				CASHCODE_STATE.RESET:
				CASHCODE_STATE.DISABLE:
					IF NOT fl_disableCashCode THEN
						eStateCashCode := CASHCODE_STATE.INIT;
					END_IF
			END_CASE

		CCNET_STATE.SEND_RESET:
			_BUFFER_CLEAR(PT:=ADR(sReadBuff), SIZE:=SIZEOF((sReadBuff)));
			_BUFFER_CLEAR(PT:=ADR(sReadData), SIZE:=SIZEOF((sReadData)));
			_BUFFER_CLEAR(PT:=ADR(sWriteData), SIZE:=SIZEOF((sWriteData)));
			SET_RESET();
			xDone := FALSE;
			szReadData := 0;
			eStateCCNET := CCNET_STATE.SEND_COMMAND;
		
		CCNET_STATE.SEND_POLL:
			_BUFFER_CLEAR(PT:=ADR(sReadBuff), SIZE:=SIZEOF((sReadBuff)));
			_BUFFER_CLEAR(PT:=ADR(sReadData), SIZE:=SIZEOF((sReadData)));
			_BUFFER_CLEAR(PT:=ADR(sWriteData), SIZE:=SIZEOF((sWriteData)));
			fb_COMread
			(
				xExecute := TRUE,
				hCom := hCom,
				pBuffer := ADR(sReadData),
				szBuffer := SIZEOF(sReadData),
			);
			IF  fb_COMread.xDone THEN
				szReadData1 := fb_COMread.szSize;
				fb_COMread(xExecute:=FALSE);
				IF  szReadData1 = 0 THEN 
					eStateCCNET := CCNET_STATE.SEND_COMMAND;
				END_IF
			END_IF
		
			_BUFFER_CLEAR(PT:=ADR(sReadBuff), SIZE:=SIZEOF((sReadBuff)));
			_BUFFER_CLEAR(PT:=ADR(sReadData), SIZE:=SIZEOF((sReadData)));
			_BUFFER_CLEAR(PT:=ADR(sWriteData), SIZE:=SIZEOF((sWriteData)));
			SET_POLL();
			xDone := FALSE;
			szReadData := 0;

		CCNET_STATE.SEND_ENABLE_BILL_TYPES:
			_BUFFER_CLEAR(PT:=ADR(sReadBuff), SIZE:=SIZEOF((sReadBuff)));
			_BUFFER_CLEAR(PT:=ADR(sReadData), SIZE:=SIZEOF((sReadData)));
			_BUFFER_CLEAR(PT:=ADR(sWriteData), SIZE:=SIZEOF((sWriteData)));
			SET_ENABLE_BILL_TYPES();
			xDone := FALSE;
			szReadData := 0;
			eStateCCNET := CCNET_STATE.SEND_COMMAND;

		CCNET_STATE.SEND_NSC:
			_BUFFER_CLEAR(PT:=ADR(sReadBuff), SIZE:=SIZEOF((sReadBuff)));
			_BUFFER_CLEAR(PT:=ADR(sReadData), SIZE:=SIZEOF((sReadData)));
			_BUFFER_CLEAR(PT:=ADR(sWriteData), SIZE:=SIZEOF((sWriteData)));
			SET_NSC();
			xDone := FALSE;
			szReadData := 0;
			fb_COMwrite
			(
				xExecute := TRUE,
				hCom := hCom,
				pBuffer := ADR(sWriteData),
				szSize := szWriteDataLen
				//szSize := INT_TO_UINT(LEN(sWriteData))
			);
			IF fb_COMwrite.xError THEN
				xWriteError := TRUE;
				eStateCCNET := CCNET_STATE.POLLING_CYCLE_ENDS;
			END_IF
			IF fb_COMwrite.xDone THEN
				fb_COMwrite(xExecute:=FALSE);
				xWriteError := FALSE;
				eStateCCNET := CCNET_STATE.RESPONSE_DELAY;
			END_IF

		CCNET_STATE.SEND_ASC:
			_BUFFER_CLEAR(PT:=ADR(sReadBuff), SIZE:=SIZEOF((sReadBuff)));
			_BUFFER_CLEAR(PT:=ADR(sReadData), SIZE:=SIZEOF((sReadData)));
			_BUFFER_CLEAR(PT:=ADR(sWriteData), SIZE:=SIZEOF((sWriteData)));
			SET_ACK();
			xDone := FALSE;
			szReadData := 0;
			fb_COMwrite
			(
				xExecute := TRUE,
				hCom := hCom,
				pBuffer := ADR(sWriteData),
				szSize := szWriteDataLen
				//szSize := INT_TO_UINT(LEN(sWriteData))
			);
			IF fb_COMwrite.xError THEN
				xWriteError := TRUE;
				eStateCCNET := CCNET_STATE.POLLING_CYCLE_ENDS;
			END_IF
			IF fb_COMwrite.xDone THEN
				fb_COMwrite(xExecute:=FALSE);
				xWriteError := FALSE;
				eStateCCNET := CCNET_STATE.RESPONSE_DELAY;
			END_IF
			
		CCNET_STATE.SEND_COMMAND:
			fb_COMwrite
			(
				xExecute := TRUE,
				hCom := hCom,
				pBuffer := ADR(sWriteData),
				szSize := szWriteDataLen
				//szSize := INT_TO_UINT(LEN(sWriteData))
			);
			IF fb_COMwrite.xError THEN
				xWriteError := TRUE;
				eStateCCNET := CCNET_STATE.POLLING_CYCLE_ENDS;
			END_IF
			
			fb_TON_Poll(IN:=FALSE, PT:=c_tDelay);
			fb_TON_Poll(IN:=TRUE, PT:=c_tDelay);


			IF fb_COMwrite.xDone THEN
				fb_COMwrite(xExecute:=FALSE);
				xWriteError := FALSE;
				fb_TON_Write(IN:=FALSE, PT:=c_tTimeoutWrite);
				fb_TON_Write(IN:=TRUE, PT:=c_tTimeoutWrite);
				
				fb_TON_Read(IN:=FALSE, PT:=c_tTimeoutRead);
				fb_TON_Read(IN:=TRUE, PT:=c_tTimeoutRead);
				eStateCCNET := CCNET_STATE.WAIT_WRITE;
			END_IF

		CCNET_STATE.WAIT_WRITE:
			fb_TON_Write();
			IF fb_TON_Write.Q THEN
				eStateCCNET := CCNET_STATE.RECEIVE_RESPONSE;
				fb_TON_Write(IN:=FALSE);
			END_IF
		

		CCNET_STATE.RECEIVE_RESPONSE:
			fb_COMread
			(
				xExecute := TRUE,
				hCom := hCom,
				pBuffer := ADR(sReadData),
				szBuffer := SIZEOF(sReadData),
			);
			fb_TON_Read();
			IF fb_COMread.xError THEN
				xReadError := TRUE;
				eStateCCNET := CCNET_STATE.POLLING_CYCLE_ENDS;
			END_IF
			
			IF fb_COMread.xDone THEN
				xTimeout:=FALSE;
				CHECK_RESPONSE();
				fb_COMread(xExecute:=FALSE);
				IF xCorrectAnswer THEN
					GET_DATA_FROM_RESPONSE();
					fb_TON_Read(IN:=FALSE, PT:=c_tTimeoutRead);
					IF Status.moneyReceived > 0  THEN
						eStateCCNET := CCNET_STATE.WAIT_ENROLLMENT;
						sum := sum + Status.moneyReceived;
					ELSE
						eStateCCNET := CCNET_STATE.SEND_ASC;
					END_IF
					
					
				//ELSE
				//	//SET_NSC();
				//	eStateCCNET := CCNET_STATE.SEND_NSC;
				//	fb_TON_Read(IN:=FALSE, PT:=c_tTimeout);
				END_IF
				
			END_IF
			
			
			IF fb_TON_Read.Q THEN
				xTimeout := TRUE;
				eStateCCNET := CCNET_STATE.SEND_NSC;
				fb_TON_Read(IN:=FALSE, PT:=c_tTimeoutRead);
//				OUTPUTS_TO_ZERO();
//				eStateCCNET := CCNET_STATE.RESPONSE_DELAY;
			END_IF

		CCNET_STATE.WAIT_ENROLLMENT:
			IF Status.moneyReceived  = 0 THEN
				eStateCCNET := CCNET_STATE.SEND_ASC;				
			END_IF
 			
			
			
		
		CCNET_STATE.RESPONSE_DELAY:
//			fb_TON(IN:=FALSE, PT:=c_tDelay);
//			fb_TON(IN:=TRUE, PT:=c_tDelay);
			eStateCCNET := CCNET_STATE.POLLING_CYCLE_ENDS;
			
		CCNET_STATE.POLLING_CYCLE_ENDS:
			fb_TON_Poll();
			IF fb_TON_Poll.Q THEN
				fb_COMread (xExecute:=FALSE);
				fb_COMwrite(xExecute:=FALSE);
				xCorrectAnswer := FALSE;
				xDone := TRUE;
				fb_TON_Poll(IN:=FALSE);
				eStateCCNET := CCNET_STATE.IDLE;
			END_IF

	END_CASE
	ELSE
		xDone := FALSE;
		xCorrectAnswer := FALSE;
//		OUTPUTS_TO_ZERO();
		eStateCCNET := CCNET_STATE.IDLE;
END_IF

ACTION CHECK_RESPONSE:
IF fb_COMread.szSize >= 6 THEN
//sReadData := CONCAT(sReadData,sReadBuff);
// szReadData := szReadData + fb_COMread.szSize;
 
// IF szReadData > 6 THEN
	wCRC:=GetCRC16(ADR(sReadData),UDINT_TO_WORD(fb_COMread.szSize-2) );   // Получим CRC 

	sWriteData[4] := WORD_TO_BYTE(wCRC); //LSB FIrst
	sWriteData[5] := WORD_TO_BYTE(SHR(wCRC, 8));

 	IF wCRC>0 OR (sReadData[fb_COMread.szSize-2] = WORD_TO_BYTE(wCRC) AND sReadData[fb_COMread.szSize-1] = WORD_TO_BYTE(SHR(wCRC, 8)) ) THEN
		FOR i:=0 TO UDINT_TO_INT(fb_COMread.szSize - 3) DO
			sReadBuff[i]:=sReadData[i];
		END_FOR
		xCorrectAnswer := TRUE;
	END_IF 
	 
// END_IF
 (*
     if (CRC16[0] = FAnswer[FLengthAnswer-2]) and (CRC16[1] = FAnswer[FLengthAnswer-1])
    //ответ полный и CRC верный а значит 100 % что данные верны, положим их в дату
    then
      begin
        // 5 это 1 байт синхронизации, 1 байт адресс девайса, 1 байт - длина данных, 2 байт - CRC
        CopyMemory(@FData,@FAnswer[3],FLengthAnswer-5);
        FLengthData:=FLengthAnswer-5;
      end
    else begin
           SendNSC(); // Скажем купу что мы получили неверный ответ
           raise Exception.Create('Не верный CRC ответа.');
         end;
  end

 
	IF FIND(sReadData, '>') <> 0 AND FIND(sReadData, '$R') <>0 AND
		(FIND(sReadData, '$R') > FIND(sReadData, '>')) THEN
		sReadData:=MID(sReadData, FIND(sReadData, '$R') - FIND(sReadData, '>') + 1,
		FIND(sReadData, '>'));
		xCorrectAnswer:=TRUE;
	END_IF
	*)
END_IF
END_ACTION

ACTION GET_DATA_FROM_RESPONSE:

IF eStateCashCode = CASHCODE_STATE.POLL THEN
	Z1 := sReadData[3]; //sReadData[fb_COMread.szSize-2]
	IF sReadData[2] = 7 THEN
		Z2 := sReadData[4];
	ELSE 
		Z2 := 0;	
	END_IF
	
	msg := "------";
	CASE Z1 OF
		
		16#10: //Power Up
				msg := "Power Up";
		16#11: //Power Up with Bill in Validator
				msg := "Power Up with Bill in Validator";
		16#12: // Power Up with Bill in Stacker
				msg := "Power Up with Bill in Stacker";
		16#13: //Initialize
				msg := "Initialize";
		16#14: //Idling
				msg := "Idling";
		16#15: //Accepting
				msg := "Accepting";
		16#17: //Stacking
				msg := "Stacking";
		16#18: //Returning
				msg := "Returning";
		16#19: //Unit Disabled
				msg := "Unit Disabled";
				eStateCashCode := CASHCODE_STATE.DISABLE;
		16#1A: //Holding
				msg := "Holding";
		16#1B: //Device Busy
				msg := "Device Busy";
		
		16#80: //money escrow!
				msg := "money escrow";
			cacheCodeConvertByteToMoney := 0;
			
			CASE Z2 OF
			   2: cacheCodeConvertByteToMoney :=10;
			   3: cacheCodeConvertByteToMoney :=50;
			   4: cacheCodeConvertByteToMoney :=100;
			   5: cacheCodeConvertByteToMoney :=500;
			   6: cacheCodeConvertByteToMoney :=1000;
			   7: cacheCodeConvertByteToMoney :=5000;   
			END_CASE
			
		
		16#81: //money received!
				msg := "money received";
			cacheCodeConvertByteToMoney := 0;
			
			CASE Z2 OF
			   2: cacheCodeConvertByteToMoney :=10;
			   3: cacheCodeConvertByteToMoney :=50;
			   4: cacheCodeConvertByteToMoney :=100;
			   5: cacheCodeConvertByteToMoney :=500;
			   6: cacheCodeConvertByteToMoney :=1000;
			   7: cacheCodeConvertByteToMoney :=5000;   
			END_CASE
			// счётчики по номиналам
			CASE Z2 OF
			   2: 
				   Status.receivedBanknote10 := 1;
			   3: 
				   Status.receivedBanknote50 := 1;
			   4:
					Status.receivedBanknote100 := 1; 
			   5:
					Status.receivedBanknote500 := 1; 
			   6:
					Status.receivedBanknote1000 := 1; 
			   7:
					Status.receivedBanknote5000 := 1; 
			END_CASE				
			//Status.countBanknote := 1; // +=1?
			//sum := sum + cacheCodeConvertByteToMoney;
			//amountReceived := cacheCodeConvertByteToMoney;
			Status.moneyReceived := cacheCodeConvertByteToMoney;
	
		16#1C: //Generic rejecting code.	
					msg := "Generic rejecting code.";
			CASE Z2 OF
				16#60:	// Insertion error - Rejecting due TO Insertion
					msg := "Insertion error";
				16#61:	// Rejecting due to Magnetic - Dielectric error
					msg := "Rejecting due to Magnetic";
				16#62:	// Rejecting due to Remained bill in head - Previously inserted bill remains in head
					msg := "Rejecting due to Remained bill in head";
				16#63:	// Rejecting due to Multiplying - Compensation error/multiplying factor error
					msg := "Rejecting due to Multiplying";
				16#64:	//Rejecting due to Conveying - Bill transport error
					msg := "Rejecting due to Conveying";
				16#65:	//Rejecting due to Identification1 - Identification error
					msg := "Rejecting due to Identification1";
				16#66:	//Rejecting due to Verification - Verification error
					msg := "Rejecting due to Verification";
				16#67:	//Rejecting due to Optic - Optic Sensor error
					msg := "Rejecting due to Optic";
				16#68:	//Rejecting due to Inhibit - Return by “inhibit denomination” error
					msg := "Rejecting due to Inhibit";
				16#69:	//Rejecting due to Capacity - Capacitance error
					msg := "Rejecting due to Capacity";
				16#6A:	//Rejecting due to Operation - Operation error
					msg := "Rejecting due to Operation";
				16#6C:	//Rejecting due to Length - Length error
					msg := "Rejecting due to Length";

				16#92:	//Rejecting due to unrecognised barcode - Bill taken was treated as a barcode but no reliable data can be read from it.
					msg := "Rejecting due to unrecognised barcode";

				16#6D:	//Rejecting due to UV - Banknote UV properties do not meet the predefined criteria
					msg := "Rejecting due to UV";

				16#93:	//Rejecting due to incorrect number of characters in barcode - Barcode data was read (at list partially) but is inconsistent.
					msg := "Rejecting due to incorrect number of characters in barcode";

				16#94:	//Rejecting due to unknown barcode start sequence - Barcode was not read as no synchronization was established.
					msg := "Rejecting due to unknown barcode start sequence";

				16#95:	//Rejecting due to unknown barcode stop sequence - Barcode was read but trailing data is corrupt.
					msg := "Rejecting due to unknown barcode stop sequence";
			END_CASE

		16#41: // Drop Cassette Full - Drop Cassette full condition	
				msg := "Drop Cassette Full";
				;
		16#42: // Drop Cassette out of position - The Bill Validator has detected the drop cassette to be open or removed.
				msg := "Drop Cassette out of position";
				;
		16#43: // Validator Jammed - A bill(s) has jammed in the acceptance path.	
				msg := "Validator Jammed";
		16#44: // Drop Cassette Jammed - A bill has jammed in drop cassette.	
				msg := "Drop Cassette Jammed";
				;
		16#45: // Cheated - Bill Validator sends this event if the intentions of the user to deceive the Bill Validator are detected.
				msg := "Cheated";
				;

		16#46: // Pause  - When the user tries to insert a second bill when the previous bill is in the Bill Validator but has not been stacked. 
			   // Thus Bill Validator stops motion of the second bill until the second bill is removed.*				
				msg := "Pause";
				;

		16#47: // Generic Failure codes	
			CASE Z2 OF
				16#50:	// Stack Motor Failure - Drop Cassette Motor failure
					msg := "Stack Motor Failure";
				16#51:	// Transport Motor Speed Failure
					msg := "Transport Motor Speed Failure";
				16#52:	// Transport Motor Failure
					msg := "Transport Motor Failure";
				16#53:	// Aligning Motor Failure
					msg := "Aligning Motor Failure";
				16#54:	// Initial Cassette Status Failure
					msg := "Initial Cassette Status Failure";
				16#55:	// Optic Canal Failure
					msg := "Optic Canal Failure";
				16#56:	// Magnetic Canal Failure - Inductive sensor failed to respond
					msg := "Magnetic Canal Failure";
				16#5F:	// Capacitance Canal Failure - Capacitance sensor failed to respond
					msg := "Capacitance Canal Failure";
			END_CASE
		
	END_CASE //Z1
	
	// состояние и ошибка купюрника
	CASE Z1 OF
		16#10, 16#11, 16#12, 16#13, 16#14, 16#15, 16#17, 16#18, 16#19, 16#1A, 16#1B:
			Status.cashcodeStatus := Z1;
			Status.cashcodeError := 0;
		16#1C:
			Status.cashcodeStatus := Z2;
			Status.cashcodeError := 0;
		16#41, 16#42, 16#43, 16#44, 16#45, 16#46:
			Status.cashcodeStatus := 16#FF;
			Status.cashcodeError := Z1;
		16#47:
			Status.cashcodeStatus := 16#FF;
			Status.cashcodeError := Z2;
	END_CASE
	

	// снятие кассеты
	IF Z1 = 16#42 THEN
		Status.casetteDropped := 1;
	ELSE
		Status.casetteDropped := 0;
	END_IF
		
	// замятие
	IF Z1 = 16#43 OR Z1 = 16#44 THEN
		Status.banknoteJammed := 1;
	ELSE
		Status.banknoteJammed := 0;
	END_IF
END_IF
END_ACTION

METHOD GetCRC16 : WORD
///calculate CRC for buffer; receive full command buffer
//FUNCTION cacheCodeCRC : WORD
VAR_INPUT
	iCommandBuffer: POINTER TO BYTE;
	iCommandBufferSize: WORD;
END_VAR
VAR
	i: WORD;
	tmpCRC: WORD;
	j: WORD;
END_VAR
GetCRC16 := 0;
FOR i := 0 TO iCommandBufferSize - 1 DO
	tmpCRC := GetCRC16 XOR iCommandBuffer[i];
	FOR j := 0 TO 7 DO
		IF (tmpCRC AND WORD#16#0001) <> 0 THEN
			tmpCRC := SHR (tmpCRC,1);
			tmpCRC := tmpCRC XOR WORD#16#08408;
		ELSE
			tmpCRC := SHR (tmpCRC, 1);
		END_IF
	END_FOR;
	GetCRC16 := tmpCRC;	
END_FOR
END_METHOD

ACTION SET_ACK:
(*
sWriteData[0]:=16#23;
sAdress:=BYTE_TO_STRH(byAdress);
sWriteData[1]:=sAdress[0];
sWriteData[2]:=sAdress[1];
byCRC:=sWriteData[0]+sWriteData[1]+sWriteData[2];
sCRC:=BYTE_TO_STRH(byCRC);
sWriteData[3]:=sCRC[0];
sWriteData[4]:=sCRC[1];
sWriteData[5]:=16#D;
*)
//ClearCommand();

  //byLengthCommand:=6;
  szWriteDataLen := 6+0; //Длина всего пакета включая CRC

  sWriteData[0] := 02; // Синхронизационный байт
  sWriteData[1] := 03; // Адресс валидатора
  sWriteData[2] := UDINT_TO_BYTE(szWriteDataLen); //Длина всего пакета включая CRC
  sWriteData[3] := 16#00;   // Команда

  wCRC:=GetCRC16(ADR(sWriteData),UDINT_TO_WORD(szWriteDataLen-2) );   // Получим CRC
  sWriteData[4] := WORD_TO_BYTE(wCRC); //LSB FIrst
  sWriteData[5] := WORD_TO_BYTE(SHR(wCRC, 8));
  
(*
cacheCodeGetNoDataCommandBuffer[0] := BYTE#16#02; //Sync
cacheCodeGetNoDataCommandBuffer[1] := iPeripheralAddress; 
cacheCodeGetNoDataCommandBuffer[2] := BUFFER_SIZE; //full data length with crc 
cacheCodeGetNoDataCommandBuffer[3] := iCommandCode;

crc:=cacheCodeCrc(iCommandBuffer := ADR(cacheCodeGetNoDataCommandBuffer), iCommandBufferSize := BUFFER_SIZE);
cacheCodeGetNoDataCommandBuffer[4] := WORD_TO_BYTE(crc); //LSB FIrst
cacheCodeGetNoDataCommandBuffer[5] := WORD_TO_BYTE(SHR(crc, 8));
*)
  
//  if Length(Data) <> 0 // Если есть данные для пеердачи
//  then CopyMemory(@FCommand[4],@Data,Length(Data)); // Скопируем их все начиная с 5 байта
(*
  wCRC:=GetCRC16(sWriteData,6-2);   // Получим CRC
  CopyMemory(@CRC16,@CRCWord,2);             // Разабьем CRC на байты

  FCommand[FLengthCommand-2]:=CRC16[0];           // Подпишем нашу команду
  FCommand[FLengthCommand-1]:=CRC16[1];
*)
END_ACTION

ACTION SET_ENABLE_BILL_TYPES:
  szWriteDataLen := 6+6; //Длина всего пакета включая CRC

  sWriteData[0] := 02; // Синхронизационный байт
  sWriteData[1] := 03; // Адресс валидатора
  sWriteData[2] := UDINT_TO_BYTE(szWriteDataLen); //Длина всего пакета включая CRC
  sWriteData[3] := 16#34;   // Команда

  // примаемые купюры
  sWriteData[4] := 2#0000_0000;   // 
  sWriteData[5] := 2#0000_0000;   // 
  sWriteData[6] := 2#0001_1000;   //
  // депонируемые купюры (отложенные)
  sWriteData[7] := 2#1111_1111;   // 
  sWriteData[8] := 2#1111_1111;   // 
  sWriteData[9] := 2#1110_0111;   // 

  wCRC:=GetCRC16(ADR(sWriteData),UDINT_TO_WORD(szWriteDataLen-2) );   // Получим CRC
  sWriteData[10] := WORD_TO_BYTE(wCRC); //LSB FIrst
  sWriteData[11] := WORD_TO_BYTE(SHR(wCRC, 8));
END_ACTION

ACTION SET_NSC:
  szWriteDataLen := 6+0; //Длина всего пакета включая CRC

  sWriteData[0] := 02; // Синхронизационный байт
  sWriteData[1] := 03; // Адресс валидатора
  sWriteData[2] := UDINT_TO_BYTE(szWriteDataLen); //Длина всего пакета включая CRC
  sWriteData[3] := 16#FF;   // Команда

  wCRC:=GetCRC16(ADR(sWriteData),UDINT_TO_WORD(szWriteDataLen-2) );   // Получим CRC
  sWriteData[4] := WORD_TO_BYTE(wCRC); //LSB FIrst
  sWriteData[5] := WORD_TO_BYTE(SHR(wCRC, 8));
END_ACTION

ACTION SET_PAKET:

END_ACTION

ACTION SET_POLL:
  szWriteDataLen := 6+0; //Длина всего пакета включая CRC

  sWriteData[0] := 02; // Синхронизационный байт
  sWriteData[1] := 03; // Адресс валидатора
  sWriteData[2] := UDINT_TO_BYTE(szWriteDataLen); //Длина всего пакета включая CRC
  sWriteData[3] := 16#33;   // Команда

  wCRC:=GetCRC16(ADR(sWriteData),UDINT_TO_WORD(szWriteDataLen-2) );   // Получим CRC
  sWriteData[4] := WORD_TO_BYTE(wCRC); //LSB FIrst
  sWriteData[5] := WORD_TO_BYTE(SHR(wCRC, 8));
END_ACTION

ACTION SET_RESET:
  szWriteDataLen := 6+0; //Длина всего пакета включая CRC

  sWriteData[0] := 02; // Синхронизационный байт
  sWriteData[1] := 03; // Адресс валидатора
  sWriteData[2] := UDINT_TO_BYTE(szWriteDataLen); //Длина всего пакета включая CRC
  sWriteData[3] := 16#30;   // Команда

  wCRC:=GetCRC16(ADR(sWriteData),UDINT_TO_WORD(szWriteDataLen-2) );   // Получим CRC
  sWriteData[4] := WORD_TO_BYTE(wCRC); //LSB FIrst
  sWriteData[5] := WORD_TO_BYTE(SHR(wCRC, 8));

 // sWriteData[4] := 65;   // 
 // sWriteData[5] := 179;   //
END_ACTION

METHOD resetMoneyReceived : word
VAR_INPUT
END_VAR
Status.moneyReceived := 0;
END_METHOD

METHOD resetMoneyCnt
VAR_INPUT
END_VAR
Status.receivedBanknote10 := 0;
Status.receivedBanknote50 := 0;
Status.receivedBanknote100 := 0; 
Status.receivedBanknote500 := 0; 
Status.receivedBanknote1000 := 0; 
Status.receivedBanknote5000 := 0;
END_METHOD

END_FUNCTION_BLOCK

// CompWin/AppTerminalPost/Cash/_BUFFER_CLEAR
FUNCTION _BUFFER_CLEAR : BOOL
VAR_INPUT
	PT : POINTER TO BYTE;
	SIZE : UINT;
END_VAR

VAR
	ptw : POINTER TO DWORD;
	temp: DWORD;
	end, end32 : DWORD;
END_VAR

temp := pt;
end := temp + UINT_TO_DWORD(size);
end32 := end - 3;
WHILE (pt < end) AND ((temp AND 16#00000003) > 0) DO
pt^ := 0;
pt := pt + 1;
temp := temp + 1;
END_WHILE;
ptw := pt;
WHILE ptw < end32 DO
ptw^ := 0;
ptw := ptw + 4;
END_WHILE;
pt := ptw;
WHILE pt < end DO
pt^ := 0;
pt := pt + 1;
END_WHILE;
_BUFFER_CLEAR := TRUE;

END_FUNCTION

// CompWin/AppTerminalPost/Cash/ANALYZE_DATA
FUNCTION_BLOCK ANALYZE_DATA
VAR_INPUT
sData: STRING;
END_VAR
VAR CONSTANT
c_iMaxCanal: INT := 8;
END_VAR
VAR_OUTPUT
arValue: ARRAY [1..c_iMaxCanal] OF REAL;
END_VAR
VAR
aiSignPos: ARRAY [1..c_iMaxCanal+1] OF INT;
i,j: INT;
END_VAR

j:=1;
FOR i:=1 TO FIND(sData,'$R') DO
IF sData[i]=16#2B OR sData[i]=16#2D OR sData[i]=16#0D THEN
aiSignPos[j]:=i;
j:=j+1;
END_IF
END_FOR
FOR i:=1 TO c_iMaxCanal-1 DO
arValue[i]:= STRING_TO_REAL(MID(sData, aiSignPos[i+1] - aiSignPos[i], aiSignPos[i] + 1));
END_FOR
arValue[c_iMaxCanal]:=STRING_TO_REAL(
MID(sData, aiSignPos[c_iMaxCanal+1] - aiSignPos[c_iMaxCanal] - 2,
aiSignPos[i] + 1));

END_FUNCTION_BLOCK

// CompWin/AppTerminalPost/Cash/BYTE_TO_STRH
FUNCTION BYTE_TO_STRH : STRING(2)
VAR_INPUT
IN : BYTE;
END_VAR
VAR
temp : BYTE;
PT : POINTER TO BYTE;
END_VAR

PT := ADR(BYTE_TO_STRH);
temp := SHR(in,4);
IF temp <= 9 THEN temp := temp + 48; ELSE temp := temp + 55; END_IF;
PT^ := temp;
temp := in AND 2#00001111;
IF temp <= 9 THEN temp := temp + 48; ELSE temp := temp + 55; END_IF;
pt := pt + 1;
pt^ := temp;
pt := pt + 1;
pt^:= 0;

END_FUNCTION

// CompWin/AppTerminalPost/DevCoin/DeviceCoin
PROGRAM DeviceCoin
VAR
	amountReceived : WORD :=0;	
	_amountReceivedTemp: WORD := 0;

	_device: ccTalk;
	_deviceStatus: ccTalkStatus;
	_isInitialized: BOOL := FALSE;

	_isCollected: BOOL := FALSE;	// Признак проведённой инкассации для сброса количества купюр
//	countCoin: UINT := 0;		// Количество купюр в боксе

	uWarningCountCoin:		UINT;	//Предупредительное	количество монет в	приёмнике (шт)
	uMAXCountCoin:			UINT;	//Максимальное кол-во монет в CashBox (шт)

	message: STRING;
END_VAR

//В самом начале с помощью метода init задаём конфигурацию модуля
//Это делается один раз
IF NOT (_isInitialized) THEN
// инициализация монетника
//	_device.init(iComPort:= 3, iCoinTypes :=  COIN_10RUB OR COIN_5RUB OR COIN_2RUB OR COIN_1RUB);
	_device.init(iComPort:= 3, iCoinTypes :=  COIN_10RUB);
	_isInitialized :=  TRUE;
END_IF;

//проводим итерацию рабочего цикла и узнаём новый статус блока
_deviceStatus:=_device.iterateAndUpdateStatus();

IF (_deviceStatus.error = CCTALK_NO_ERROR AND NOT (_deviceStatus.busy) AND _deviceStatus.moneyReceived > 0) THEN
//	totalMoneyReceived := totalMoneyReceived + ccTalkStatus.moneyReceived;
	_amountReceivedTemp := _amountReceivedTemp + _deviceStatus.moneyReceived;
	//countCoin := countCoin + _deviceStatus.countCoin;

	PersistentVars.counterCoin10 := PersistentVars.counterCoin10 + _deviceStatus.receivedCoin10;

	// увеличить тотальные счётчики номиналов
	PersistentVars.totalCoin10 := PersistentVars.totalCoin10 + _deviceStatus.receivedCoin10;
END_IF

// если внешней программой была обработана сумма, то перенести принятую сумму в прееменную для внешенй обработки
IF(amountReceived = 0 AND _amountReceivedTemp > 0)THEN
	amountReceived := _amountReceivedTemp;
	_amountReceivedTemp := 0;
END_IF

// если внешней программой был сброшен счётчик купюр, то сбросить его внутри
IF(_isCollected)THEN
	//countCoin := 0;
(*	// Coin: m1=7; m2=8; m5=9; m10=10;
	message := 'Coin: ';
	message := CONCAT(message, 'm1=');
	message := CONCAT(message, WORD_TO_STRING(DeviceCoin.GetCounterCoin(1)));
	message := CONCAT(message, '; ');
	
	message := CONCAT(message, 'm2=');
	message := CONCAT(message, WORD_TO_STRING(DeviceCoin.GetCounterCoin(2)));
	message := CONCAT(message, '; ');
	
	message := CONCAT(message, 'm5=');
	message := CONCAT(message, WORD_TO_STRING(DeviceCoin.GetCounterCoin(5)));
	message := CONCAT(message, '; ');
	
	message := CONCAT(message, 'm10=');
	message := CONCAT(message, WORD_TO_STRING(DeviceCoin.GetCounterCoin(10)));
	message := CONCAT(message, ';');
	
	PersistentVars.messageCollectCoin := message;
*)

	// запомнить значения счётчиков
	// только если было начало инкассации и счётчики ещё не сброшены
	// (защита от повторного нажатия кнопок инкассации)
	IF(PersistentVars.counterBefCollectCoin10 = 0) THEN
		PersistentVars.counterBefCollectCoin10 := PersistentVars.counterCoin10;
	END_IF
		
	// сбросить значения
	PersistentVars.counterCoin10 := 0;

	_isCollected := FALSE;
END_IF

// Вернуть во вне принятую сумму, 
// затем сбросить сумму для записывания следующих принятий
METHOD PUBLIC GetReceived : WORD
GetReceived := amountReceived;

amountReceived := 0;
END_METHOD

METHOD PUBLIC DbgInCoin : BYTE
VAR_INPUT
END_VAR
VAR
	received: WORD := 0;
END_VAR
received := DBG_PRG.GetInCoin();
IF(received > 0)THEN
	_amountReceivedTemp := _amountReceivedTemp + received;
	//countCoin := countCoin + 1;
END_IF
END_METHOD

METHOD PUBLIC CollectCash : UINT
VAR_INPUT
END_VAR
// выстаитьВыставить признка необходимости сброса счётчика монет
_isCollected := TRUE;
END_METHOD

METHOD GetCounterCoin : UINT
VAR_INPUT
	// номинал
	nom: INT;
END_VAR
GetCounterCoin := 0;

CASE nom OF
	0:
		GetCounterCoin := PersistentVars.counterCoin10;
	10:
		GetCounterCoin := PersistentVars.counterCoin10;
END_CASE
END_METHOD

END_PROGRAM

// CompWin/AppTerminalPost/DevCoin/ccTalk
FUNCTION_BLOCK ccTalk
VAR CONSTANT
//	COM_PORT : BYTE := 2;  //use com2
	CCTALK_SLAVE_ID : BYTE := 2; //destination id
	CCTALK_MASTER_ID :BYTE := 1;
	
	CCTALK_COMMAND_RESET : BYTE := 1;  //reset command id
	
	CCTALK_COMMAND_MODIFY_INHIBIT_STATUS : BYTE :=  231; // modify inhibit status command id

	
	CCTALK_COMMAND_MODIFY_MASTER_INHIBIT_STATUS : BYTE :=  228; // modify inhibit status command id
	MODIFY_MASTER_INHIBIT_STATUS_COMMAND_DATA : ARRAY[0..0] OF BYTE := [1];
	
	//program states
	CCTALK_INIT_STATE : BYTE :=0;
	CCTALK_FATAL_ERROR_STATE : BYTE :=1;
	CCTALK_DONE_STATE : BYTE :=2;
	CCTALK_RESET_STATE : BYTE :=3;
	CCTALK_POLL_STATE: BYTE :=4;
	CCTALK_WAIT_STATE : BYTE :=5;
	CCTALK_DO_NOTHING_STATE: BYTE :=6;
	CCTALK_MODIFY_INHIBIT_STATUS_STATE: BYTE :=7;
	CCTALK_MODIFY_MASTER_INHIBIT_STATUS_STATE: BYTE :=8;
	CCTALK_READ_BUFFERED_CREDIT_STATE: BYTE :=9;
	
	CCTALK_CLOSE_COM_STATE : BYTE :=10;
	

END_VAR


VAR	

	RESET_TRYCOUNT_DELAY : TIME := T#1000MS; //delay between reset tries	
	POLL_DELAY : TIME := T#200MS;

	//cachecode program states
	state : BYTE := CCTALK_INIT_STATE;
	
	error: CCTALK_ERROR := CCTALK_INIT_PROC_NOT_CALLED;
	
	
	
	//com parameters
	ccTalkComParams : ARRAY [1..7] OF COM.PARAMETER := [     
		(udiParameterId := COM.CAA_Parameter_Constants.udiPort, udiValue := 0),  // COM порт
		(udiParameterId := COM.CAA_Parameter_Constants.udiBaudrate, udiValue := 9600),
		(udiParameterId := COM.CAA_Parameter_Constants.udiParity,udiValue := INT_TO_UDINT(COM.PARITY.NONE)),
	    (udiParameterId := COM.CAA_Parameter_Constants.udiStopBits,udiValue := INT_TO_UDINT(COM.STOPBIT.ONESTOPBIT)),
		(udiParameterId := COM.CAA_Parameter_Constants.udiTimeout, udiValue := 0),
		(udiParameterId := COM.CAA_Parameter_Constants.udiByteSize, udiValue := 8),
		(udiParameterId := COM.CAA_Parameter_Constants.udiBinary,udiValue := 0)
	];
	
	ccTalkOpen : COM.Open;
	ccTalkClose : COM.Close;
	openedHCom : CAA.HANDLE := 0;
	portOpened : BOOL := FALSE;
	
	simpleCommand : ccTalkSimpleCommand;
	readBufferedCreditCommand : ccTalkReadBufferedCreditCommand;

	
	
	waitTimer : TON;

	
	test:BYTE:=2;
	
	modifyInhibitStatusCommandData : ARRAY[0..1] OF BYTE ;
	
	moneyReceived : UINT := 0;
	coinsRejected : UINT := 0;
	
	receivedCoin1  : UINT := 0;
	receivedCoin2  : UINT := 0;
	receivedCoin5  : UINT := 0;
	receivedCoin10 : UINT := 0;
	// количество монет в боксе
	countCoin: UINT := 0;	
	
	
	b_cctalk_close_enable:  BOOL := FALSE;
END_VAR

METHOD init
VAR_INPUT
	iComPort: BYTE;
	///or`d  enabled coin types
	iCoinTypes: UINT := 0;
END_VAR
//init method called -> reset error flags
state := CCTALK_INIT_STATE;
error := CCTALK_NO_ERROR;

ccTalkComParams[1].udiValue := iComPort;
modifyInhibitStatusCommandData[0] := UINT_TO_BYTE(SHR(iCoinTypes, 8));
modifyInhibitStatusCommandData[1] := UINT_TO_BYTE(iCoinTypes);
END_METHOD

METHOD iterateAndUpdateStatus : ccTalkStatus
//waiting between cycle
	
coinsRejected := 0;
moneyReceived :=0;
countCoin := 0;

receivedCoin1 := 0;
receivedCoin2 := 0;
receivedCoin5 := 0;
receivedCoin10 := 0;

IF waitTimer.IN  THEN
	waitTimer(IN:= TRUE);
	IF NOT (waitTimer.Q) THEN
		iterateAndUpdateStatus.busy := simpleCommand.xExecute OR readBufferedCreditCommand.xExecute;
		iterateAndUpdateStatus.error := error;
		iterateAndUpdateStatus.moneyReceived := moneyReceived;
		iterateAndUpdateStatus.coinsRejected := coinsRejected ;
		
		iterateAndUpdateStatus.receivedCoin1 := receivedCoin1;
		iterateAndUpdateStatus.receivedCoin2 := receivedCoin2;
		iterateAndUpdateStatus.receivedCoin5 := receivedCoin5;
		iterateAndUpdateStatus.receivedCoin10 := receivedCoin10;
		
		
		RETURN;
	ELSE
		waitTimer(IN:=FALSE);	
	END_IF
END_IF


CASE state OF
	CCTALK_INIT_STATE:
		ccTalkOpen (xExecute := TRUE, 
				usiListLength := UINT_TO_USINT(SIZEOF(ccTalkComParams)/SIZEOF(COM.PARAMETER)),
				pParameterList:= ADR(ccTalkComParams)			
		);
		openedHCom := ccTalkOpen.hCom;
		IF ccTalkOpen.xError THEN
			ccTalkOpen (xExecute := FALSE);
			portOpened := FALSE;
			state := CCTALK_FATAL_ERROR_STATE;  
			error := CCTALK_OPEN_ERROR;
		END_IF;
		
		IF ccTalkOpen.xDone THEN
			ccTalkOpen (xExecute := FALSE);
			portOpened := TRUE;
			state := CCTALK_RESET_STATE;
			error := CCTALK_NO_ERROR;
		END_IF;
	CCTALK_RESET_STATE:
		simpleCommand(xExecute:=TRUE, hCom := openedHCom, xSourceId := CCTALK_MASTER_ID, 
					xDestinationId := CCTALK_SLAVE_ID, xCommand:=CCTALK_COMMAND_RESET, xCommandDataSize:=0 );
		
		IF simpleCommand.xDone THEN
			state := CCTALK_MODIFY_INHIBIT_STATUS_STATE;
			waitTimer(IN:= TRUE, PT := POLL_DELAY);
		END_IF
		
		//retry reset
		IF simpleCommand.xError THEN   
			state := CCTALK_CLOSE_COM_STATE;
			//state := CCTALK_RESET_STATE;
			waitTimer(IN:= TRUE, PT := RESET_TRYCOUNT_DELAY);
		END_IF
	CCTALK_CLOSE_COM_STATE:
		state := CCTALK_RESET_STATE;
		IF b_cctalk_close_enable THEN
			IF portOpened THEN
			  ccTalkClose(xExecute:=TRUE, hCom := openedHCom);
			  IF ccTalkClose.xError THEN
				portOpened := FALSE;
				ccTalkClose(xExecute:=FALSE);
				state := CCTALK_INIT_STATE;  
				error := CCTALK_OPEN_ERROR;
			  END_IF;
			  IF ccTalkClose.xDone THEN
				portOpened := FALSE;
				ccTalkClose(xExecute:=FALSE);
				state := CCTALK_INIT_STATE;
			  END_IF;
			ELSE		  
				state := CCTALK_INIT_STATE;
			END_IF;
	
		END_IF

	
	CCTALK_MODIFY_INHIBIT_STATUS_STATE: //enable coin types
		simpleCommand(xExecute:=TRUE, hCom := openedHCom, xSourceId := CCTALK_MASTER_ID, 
					 xDestinationId := CCTALK_SLAVE_ID, xCommand:=CCTALK_COMMAND_MODIFY_INHIBIT_STATUS, xCommandData:=
					 ADR(modifyInhibitStatusCommandData), xCommandDataSize := UINT_TO_BYTE(SIZEOF(modifyInhibitStatusCommandData))
					);
		
		IF simpleCommand.xDone THEN
			state := CCTALK_MODIFY_MASTER_INHIBIT_STATUS_STATE;
		END_IF
		
		//retry reset
		IF simpleCommand.xError THEN    
			state := CCTALK_RESET_STATE;
			waitTimer(IN:= TRUE, PT := POLL_DELAY);
		END_IF

	CCTALK_MODIFY_MASTER_INHIBIT_STATUS_STATE: //enable master inhibit
		simpleCommand(xExecute:=TRUE, hCom := openedHCom, xSourceId := CCTALK_MASTER_ID, 
					 xDestinationId := CCTALK_SLAVE_ID, xCommand:=CCTALK_COMMAND_MODIFY_MASTER_INHIBIT_STATUS, xCommandData:=
					 ADR(MODIFY_MASTER_INHIBIT_STATUS_COMMAND_DATA), xCommandDataSize := UINT_TO_BYTE(SIZEOF(MODIFY_MASTER_INHIBIT_STATUS_COMMAND_DATA))
					);
		
		IF simpleCommand.xDone THEN
			state := CCTALK_READ_BUFFERED_CREDIT_STATE;
		END_IF
		
		//retry reset
		IF simpleCommand.xError THEN    
			state := CCTALK_RESET_STATE;
			waitTimer(IN:= TRUE, PT := POLL_DELAY);
		END_IF	

	CCTALK_READ_BUFFERED_CREDIT_STATE: //
		readBufferedCreditCommand(xExecute:=TRUE, hCom := openedHCom, xSourceId := CCTALK_MASTER_ID, 
					 xDestinationId := CCTALK_SLAVE_ID);
		
		IF readBufferedCreditCommand.xDone THEN
			moneyReceived :=  readBufferedCreditCommand.xMoneyAccepted;
			coinsRejected := readBufferedCreditCommand.xCoinsRejected;
			countCoin := readBufferedCreditCommand.xCoinsAccepted;
			
			receivedCoin1 := readBufferedCreditCommand.xReceivedCoin1;
			receivedCoin2 := readBufferedCreditCommand.xReceivedCoin2;
			receivedCoin5 := readBufferedCreditCommand.xReceivedCoin5;
			receivedCoin10 := readBufferedCreditCommand.xReceivedCoin10;
			
			state := CCTALK_READ_BUFFERED_CREDIT_STATE;
			waitTimer(IN:= TRUE, PT := POLL_DELAY);
		END_IF
		
		//retry reset
		IF readBufferedCreditCommand.xError THEN    
			state := CCTALK_RESET_STATE;
			waitTimer(IN:= TRUE, PT := POLL_DELAY);
		END_IF			
		

	
	
	CCTALK_FATAL_ERROR_STATE:
		state := CCTALK_CLOSE_COM_STATE;
	
//	CCTALK_DONE_STATE:  //all work is done, free resources
//		ccTalkOpen(xExecute := FALSE);
//		state := CCTALK_DO_NOTHING_STATE;
//						
//	CCTALK_DO_NOTHING_STATE:
END_CASE


iterateAndUpdateStatus.busy := simpleCommand.xExecute OR readBufferedCreditCommand.xExecute;
iterateAndUpdateStatus.error := error;
iterateAndUpdateStatus.moneyReceived := moneyReceived;
iterateAndUpdateStatus.coinsRejected := coinsRejected ;

iterateAndUpdateStatus.countCoin := countCoin;
iterateAndUpdateStatus.receivedCoin1 := receivedCoin1;
iterateAndUpdateStatus.receivedCoin2 := receivedCoin2;
iterateAndUpdateStatus.receivedCoin5 := receivedCoin5;
iterateAndUpdateStatus.receivedCoin10 := receivedCoin10;
END_METHOD

END_FUNCTION_BLOCK

// CompWin/AppTerminalPost/DevCoin/ccTalkSimpleCommand
///command with  no-data ack
FUNCTION_BLOCK ccTalkSimpleCommand
VAR CONSTANT
	STATE_INITIAL: BYTE := 0;
	STATE_WAIT_ACK: BYTE := 1;
	STATE_FATAL_ERROR: BYTE := 3;
	COMMAND_EXPECTED_ANSWER_SIZE: BYTE := 5;
	///maximum size of command data 
	COMMAND_DATA_SIZE_MAX: BYTE := 5;
	COMMAND_DATA_OFFSET: BYTE := 4;
	///? 
END_VAR
VAR_INPUT
	hCom: CAA.HANDLE;
	xExecute: BOOL := FALSE;
	///device address
	xDestinationId: BYTE := 2;
	///master address, default = 1;
	xSourceId: BYTE := 1;
	xCommand: BYTE;
	xCommandData: POINTER TO BYTE;
	xCommandDataSize: BYTE := 0;
END_VAR
VAR_OUTPUT
	xDone: BOOL := FALSE;
	xError: BOOL := FALSE;
	xTimeout: BOOL := FALSE;
END_VAR
VAR
	TIMEOUT: TIME := TIME#200MS;
	///buffer for command
	commandBuffer: ARRAY[0..(4 + COMMAND_DATA_SIZE_MAX)] OF BYTE;
	///size enough for echo and answer
	//readBuffer: ARRAY[0..((4 + COMMAND_DATA_SIZE_MAX) + COMMAND_EXPECTED_ANSWER_SIZE)] OF BYTE;
	readBuffer: ARRAY[0..255] OF BYTE;
	///timeout timer (timeout value - ????)
	waitingACKtimeout: TON;
	localState: BYTE := STATE_INITIAL;
	ccTalkCodeWrite: COM.Write;
	ccTalkCodeRead: COM.Read;
	bufferReaded: CAA.SIZE := 0;
	bufferFullLen: BYTE := 5;
	///full answer size with echo
	fullAnswerSize: BYTE;
	commandCode: INT;
	crc: BYTE;
END_VAR

CASE localState OF 
	STATE_INITIAL:
		IF xExecute THEN
			xDone := FALSE;
			xError := FALSE;
			xTimeout := FALSE;
			IF NOT ccTalkCodeWrite.xExecute THEN
				bufferFullLen := 5 + xCommandDataSize;
				fullAnswerSize := bufferFullLen + COMMAND_EXPECTED_ANSWER_SIZE;
				commandBuffer[0] := xDestinationId;
				commandBuffer[1] := xCommandDataSize; //data size 
				commandBuffer[2] := xSourceId;  // master address
				commandBuffer[3] := xCommand; //command code
				IF xCommandDataSize > 0 THEN
					MEM.MemMove(pSource := xCommandData, pDestination := ADR(commandBuffer) + COMMAND_DATA_OFFSET, uiNumberOfBytes := xCommandDataSize);
				END_IF;
				commandBuffer[bufferFullLen - 1] := ccTalkCRC(ADR(commandBuffer), bufferFullLen); //command code
			END_IF
			ccTalkCodeWrite(xExecute := TRUE,hCom:= hCom, pBuffer:= ADR(commandBuffer), szSize:= bufferFullLen);
			IF ccTalkCodeWrite.xError THEN
				xError := TRUE;
				xExecute := FALSE;
				xCommandDataSize :=0;
				localState := STATE_INITIAL;
				ccTalkCodeWrite(xExecute := FALSE);
				RETURN;
			END_IF
		
			// if the writing process is completed the reading process can be started
			IF ccTalkCodeWrite.xDone THEN
				localState := STATE_WAIT_ACK;
				bufferReaded := 0;
				xCommandDataSize :=0;
				ccTalkCodeWrite(xExecute := FALSE);
				waitingACKtimeout(IN:=FALSE); 
				waitingACKtimeout(IN:=TRUE, PT:=TIMEOUT);  //timeout value ?
			END_IF			
		END_IF
		//waiting ACK
	STATE_WAIT_ACK:
		waitingACKtimeout(IN:=TRUE, PT:=TIMEOUT);  //timeout value ?
		IF waitingACKTimeout.Q THEN  //timeout is over..
			xError := TRUE;
			xExecute := FALSE;
			xTimeout := TRUE;
			localState := STATE_INITIAL;
			ccTalkCodeRead(xExecute := FALSE);
		ELSE
			ccTalkCodeRead(xExecute := TRUE,hCom:= hCom, pBuffer:= ADR(readBuffer) + bufferReaded, szBuffer:= SIZEOF(readBuffer)- bufferReaded);
			IF ccTalkCodeRead.xError THEN
				xError := TRUE;
				xExecute := FALSE;
				ccTalkCodeRead(xExecute := FALSE);
				localState := STATE_INITIAL;
			END_IF
			//After completion the size of the written bytes are saved
			IF 	ccTalkCodeRead.xDone THEN
				bufferReaded := bufferReaded + ccTalkCodeRead.szSize;
				IF bufferReaded >= fullAnswerSize THEN  //try to recognize command
					//MEM.MemMove(pSource:=ADR(readBuffer) + bufferFullLen, pDestination:=ADR(readBuffer), uiNumberOfBytes:=COMMAND_EXPECTED_ANSWER_SIZE); //move data to begin
					ccTalkCodeRead(xExecute := FALSE);
					crc := ccTalkCRC(iCommandBuffer := ADR(readBuffer), iCommandBufferSize:=COMMAND_EXPECTED_ANSWER_SIZE);
					//ALL OK
					IF (crc = readBuffer[COMMAND_EXPECTED_ANSWER_SIZE -1]) THEN
						//ack format :  [ destination, 0, source, 0, crc ] 
						IF readBuffer[0] = xSourceId AND readBuffer[1] = 0 AND readBuffer[2] = xDestinationId AND readBuffer[3] = 0 THEN 
							xExecute := FALSE;
							xDone := TRUE;
							localState := STATE_INITIAL;
						ELSE 
							bufferReaded := 0;  //try to wait buffer with proper fields
						END_IF
					ELSE
						xError := TRUE;
						xExecute := FALSE;
						localState := STATE_INITIAL;
					END_IF

				END_IF

			END_IF			
		END_IF
		
END_CASE

END_FUNCTION_BLOCK

// CompWin/AppTerminalPost/DevCoin/ccTalkCRC
///calculate CRC for buffer; receive full command buffer
FUNCTION ccTalkCRC : BYTE
VAR_INPUT
	iCommandBuffer: POINTER TO BYTE;
	iCommandBufferSize: WORD;
END_VAR
VAR
	i: WORD;
END_VAR

ccTalkCRC := 0;
FOR i := 0 TO iCommandBufferSize - 2 DO
	ccTalkCrc := ccTalkCrc + iCommandBuffer[i];
END_FOR
ccTalkCRC:= 255 - ccTalkCRC;
ccTalkCRC:=ccTalkCRC + 1;

END_FUNCTION

// CompWin/AppTerminalPost/DevCoin/ccTalkReadBufferedCreditCommand
///ReadBufferedCreditCommand (229).
FUNCTION_BLOCK ccTalkReadBufferedCreditCommand
VAR CONSTANT
	STATE_INITIAL: BYTE := 0;
	STATE_WAIT_ACK: BYTE := 1;
	STATE_FATAL_ERROR: BYTE := 3;
	COMMAND_EXPECTED_ANSWER_SIZE: BYTE := 16;
	COMMAND_EXPECTED_DATA_SIZE: BYTE := 11;
	///? 
	TIMEOUT: TIME := TIME#200ms;
END_VAR
VAR_INPUT
	hCom: CAA.HANDLE;
	xExecute: BOOL := FALSE;
	///device address
	xDestinationId: BYTE := 2;
	///master address, default = 1;
	xSourceId: BYTE := 1;
END_VAR
VAR_OUTPUT
	xDone: BOOL := FALSE;
	xError: BOOL := FALSE;
	xTimeout: BOOL := FALSE;
	///Total events since reset
	xEvents: BYTE := 0;
	xEventsTable: ARRAY[0..5] OF ccTalkEvent;
	///Money accepted since last poll
	xMoneyAccepted: BYTE := 0;
	///Coins rejected since last poll
	xCoinsRejected: BYTE := 0;
	///Coins accepted since last poll
	xCoinsAccepted : BYTE :=0;
	
	//Coins 1 ruble accepted since last poll
	xReceivedCoin1 : BYTE := 0;
	//Coins 2 ruble accepted since last poll
	xReceivedCoin2 : BYTE := 0;
	//Coins 5 ruble accepted since last poll
	xReceivedCoin5 : BYTE := 0;
	//Coins 10 ruble accepted since last poll
	xReceivedCoin10 : BYTE := 0;
END_VAR
VAR
	///last events
	lastEvents: BYTE := 0;
	///buffer for command
	commandBuffer: ARRAY[0..4] OF BYTE;
	///size enough for echo and answer
	//readBuffer: ARRAY[0..(4 + COMMAND_EXPECTED_ANSWER_SIZE)] OF BYTE;
	readBuffer: ARRAY[0..255] OF BYTE;
	///timeout timer (timeout value - ????)
	waitingACKtimeout: TON;
	localState: BYTE := STATE_INITIAL;
	ccTalkCodeWrite: COM.Write;
	ccTalkCodeRead: COM.Read;
	bufferReaded: CAA.SIZE := 0;
	bufferFullLen: BYTE := 5;
	///full answer size with echo
	fullAnswerSize: BYTE;
	commandCode: INT;
	crc: BYTE;
END_VAR

CASE localState OF 
	STATE_INITIAL:
		IF xExecute THEN
			xDone := FALSE;
			xError := FALSE;
			xTimeout := FALSE;
			IF NOT ccTalkCodeWrite.xExecute THEN
				xMoneyAccepted := 0;
				xCoinsRejected :=0;
				xCoinsAccepted :=0;
				bufferFullLen := 5;
				
				xReceivedCoin1 := 0;
				xReceivedCoin2 := 0;
				xReceivedCoin5 := 0;
				xReceivedCoin10 := 0;
				
				
				fullAnswerSize := bufferFullLen + COMMAND_EXPECTED_ANSWER_SIZE;
				commandBuffer[0] := xDestinationId;
				commandBuffer[1] := 0; //data size 
				commandBuffer[2] := xSourceId;  // master address
				commandBuffer[3] := 229; //command code
				commandBuffer[bufferFullLen - 1] := ccTalkCRC(ADR(commandBuffer), bufferFullLen); //command code
			END_IF
			ccTalkCodeWrite(xExecute := TRUE,hCom:= hCom, pBuffer:= ADR(commandBuffer), szSize:= bufferFullLen);
			IF ccTalkCodeWrite.xError THEN
				xError := TRUE;
				xExecute := FALSE;
				localState := STATE_INITIAL;
				ccTalkCodeWrite(xExecute := FALSE);
				RETURN;
			END_IF
		
			// if the writing process is completed the reading process can be started
			IF ccTalkCodeWrite.xDone THEN
				localState := STATE_WAIT_ACK;
				bufferReaded := 0;
				ccTalkCodeWrite(xExecute := FALSE);
				waitingACKtimeout(IN:=FALSE); 
				waitingACKtimeout(IN:=TRUE, PT:=TIMEOUT);  //timeout value ?
			END_IF			
		END_IF
		//waiting ACK
	STATE_WAIT_ACK:
		waitingACKtimeout(IN:=TRUE, PT:=TIMEOUT);  //timeout value ?
		IF waitingACKTimeout.Q THEN  //timeout is over..
			xError := TRUE;
			xExecute := FALSE;
			xTimeout := TRUE;
			localState := STATE_INITIAL;
			ccTalkCodeRead(xExecute := FALSE);
		ELSE
			ccTalkCodeRead(xExecute := TRUE,hCom:= hCom, pBuffer:= ADR(readBuffer) + bufferReaded, szBuffer:= SIZEOF(readBuffer)- bufferReaded);
			IF ccTalkCodeRead.xError THEN
				xError := TRUE;
				xExecute := FALSE;
				ccTalkCodeRead(xExecute := FALSE);
				localState := STATE_INITIAL;
			END_IF
			//After completion the size of the written bytes are saved
			IF 	ccTalkCodeRead.xDone THEN
				bufferReaded := bufferReaded + ccTalkCodeRead.szSize;
				IF bufferReaded >= fullAnswerSize THEN  //try to recognize command
					//MEM.MemMove(pSource:=ADR(readBuffer) + bufferFullLen, pDestination:=ADR(readBuffer), uiNumberOfBytes:=COMMAND_EXPECTED_ANSWER_SIZE); //move data to begin
					ccTalkCodeRead(xExecute := FALSE);
					crc := ccTalkCRC(iCommandBuffer := ADR(readBuffer), iCommandBufferSize:=COMMAND_EXPECTED_ANSWER_SIZE);
					//ALL OK
					IF (crc = readBuffer[COMMAND_EXPECTED_ANSWER_SIZE -1]) THEN
						//ack format :  [ destination, 0, source, header=0, data, crc ] 
						IF readBuffer[0] = xSourceId AND readBuffer[1] = COMMAND_EXPECTED_DATA_SIZE AND readBuffer[2] = xDestinationId THEN 
							xExecute := FALSE;
							xDone := TRUE;
							localState := STATE_INITIAL;
							xEvents := readBuffer[4];
							MEM.MemMove(pSource:=ADR(readBuffer) + 5, pDestination := ADR(xEventsTable), SIZEOF(xEventsTable));
							xMoneyAccepted := xMoneyAccepted + 
									ccTalkProcessReadBufferCreditTable(iReadBufferCreditTable := ADR(xEventsTable), iLastEventsNum:=lastEvents, 
																	   iEventsNum :=xEvents, coinsRejected => xCoinsRejected, 
																	   coinsAccepted => xCoinsAccepted,
																	   receivedCoin1 => xReceivedCoin1,
																	   receivedCoin2 => xReceivedCoin2,
																	   receivedCoin5 => xReceivedCoin5,
																	   receivedCoin10 => xReceivedCoin10);

							lastEvents := xEvents;
						ELSE 
							bufferReaded := 0;  //try to wait buffer with proper fields
						END_IF
					ELSE
						xError := TRUE;
						xExecute := FALSE;
						localState := STATE_INITIAL;
					END_IF

				END_IF

			END_IF			
		END_IF
		
END_CASE

END_FUNCTION_BLOCK

// CompWin/AppTerminalPost/DevCoin/ccTalkProcessReadBufferCreditTable
///process  read buffer credit table, returns total amount of accepted money
FUNCTION ccTalkProcessReadBufferCreditTable : BYTE
VAR_INPUT
	///table to process, size 5
	iReadBufferCreditTable: POINTER TO ccTalkEvent;
	///events num in last poll
	iLastEventsNum: BYTE := 0;
	///events num in current poll
	iEventsNum: BYTE := 0;
END_VAR
VAR_OUTPUT
	coinsRejected: BYTE;
	coinsAccepted: BYTE;
	
	receivedCoin1 : BYTE;
	receivedCoin2 : BYTE;
	receivedCoin5 : BYTE;
	receivedCoin10 : BYTE;

END_VAR
VAR
	delta: BYTE;
	i: BYTE;
	acceptedMoney : BYTE;
END_VAR


//according to ccTalkPart1v4.7:

//IF events = 0 AND last events > 0 THEN error condition ( power fail AND possible lost credits )
//If delta(events) = 0 then no new credits
//If delta(events) >= 1 and delta(events) <= 5 then new credit information
//If delta(events) > 5 then error condition ( 1 or more lost credits )
ccTalkProcessReadBufferCreditTable :=0;
coinsRejected :=0;
coinsAccepted :=0;

receivedCoin1 :=0;
receivedCoin2 :=0;
receivedCoin5 :=0;
receivedCoin10 :=0;

IF (iEventsNum = 0 ) AND (iLastEventsNum > 0) THEN
	RETURN;
END_IF;

delta := iEventsNum - iLastEventsNum;

IF delta = 0 THEN
	RETURN;
ELSE
	delta := MIN(delta, 5);
	FOR i := 0 TO delta - 1 DO
		IF iReadBufferCreditTable[i].validationChannel > 0 THEN //inhibited coin, see G-13.mft ccTalk manual
		//IF iReadBufferCreditTable[i].errorCode = 1 THEN  //TODO : REMOVE IN RELEASE VERSION!!
			CASE iReadBufferCreditTable[i].validationChannel OF
//   				16#04, 16#05 : acceptedMoney :=1; receivedCoin1:=receivedCoin1 +1;
//   				16#06, 16#07 : acceptedMoney :=2; receivedCoin2:=receivedCoin2 +1;
//				16#08, 16#09: acceptedMoney :=5; receivedCoin5:=receivedCoin5 +1;
//				16#0A, 16#0B : acceptedMoney :=10; receivedCoin10:=receivedCoin10 +1;

//				16#08, 16#09 : acceptedMoney :=10; receivedCoin10:=receivedCoin10 +1;
				16#04: acceptedMoney :=10; receivedCoin10:=receivedCoin10 +1;
			ELSE
				 acceptedMoney :=0;
			END_CASE
			ccTalkProcessReadBufferCreditTable := acceptedMoney;  
			IF acceptedMoney > 0 THEN
				coinsAccepted := coinsAccepted +1;
			END_IF
		ELSE 
			coinsRejected := coinsRejected + 1;
		END_IF
	END_FOR
	
END_IF

END_FUNCTION

// CompWin/AppTerminalPost/DevButtons/DeviceButtons
PROGRAM DeviceButtons
VAR
//	Buttons : ARRAY [EnumButton.BTN_ACTIVECLEAN .. EnumButton.BTN_HELP] OF BOOL := [10(FALSE)];
	Buttons : ARRAY [1 .. 10] OF BOOL := [10(FALSE)];
	sumButtons : INT :=0;
	i: EnumButton;
	_activeButton : EnumButton := EnumButton.NONE;
	externalActiveButton :EnumButton := EnumButton.NONE;

		
	DOutPuts: BYTE :=0;
	
	Button : BYTE;
	Dinputs : BYTE;
	color: ARRAY[0..7] OF BYTE;
	status : BOOL;
	
	TON1 : TON;
	TON2 : TON;
	TON3 : TON;
	TON4 : TON;
	TON5 : TON;
	TON6 : TON;
	TON7 : TON;
	TON8 : TON;
	TON10 : TON;
	TP9 : TP;

	RS1 : SR;
	RS2 : SR;
	RS3 : SR;
	RS4 : SR;
	RS5 : SR;
	RS6 : SR;
	RS7 : SR;
	RS8 : SR;
	resetAll: BOOL;

	tTimeout : TIME :=T#50MS;
	//bDout: BYTE := 16#07;
	//bDin: BYTE;
	bStatusRead: BOOL;
	bStatusWrite: BOOL;
	
	btnStartEnable: EnumButton;
	btnStopEnable: EnumButton;
	fBtnCollectPushed: BOOL := FALSE;
	
	//Вспомогательные переменные
	udiResult: UDINT;
	udiTimeLocal : UDINT;
	timeDate: DATE_AND_TIME;
	
//	test1 : BOOL := FALSE;
//    command:STRING[256]:= 'omxplayer /home/pi/Videos/Idle.mp4';
//    res: SysCom.RTS_IEC_RESULT;

END_VAR

//bDin := UBRAIN1.bDin1;
bStatusRead := UBRAIN1.xValidRead;
bStatusWrite := UBRAIN1.xValidRead;

TON1(IN:=(EXTRACT(X:=UBRAIN1.bButtons, N:=0) AND UBRAIN1.xValidRead), PT:=tTimeout);
TON2(IN:=(EXTRACT(X:=UBRAIN1.bButtons, N:=1) AND UBRAIN1.xValidRead), PT:=tTimeout);
TON3(IN:=(EXTRACT(X:=UBRAIN1.bButtons, N:=2) AND UBRAIN1.xValidRead), PT:=tTimeout);
TON4(IN:=(EXTRACT(X:=UBRAIN1.bButtons, N:=3) AND UBRAIN1.xValidRead), PT:=tTimeout);
TON5(IN:=(EXTRACT(X:=UBRAIN1.bButtons, N:=4) AND UBRAIN1.xValidRead), PT:=tTimeout);
TON6(IN:=(EXTRACT(X:=UBRAIN1.bButtons, N:=5) AND UBRAIN1.xValidRead), PT:=tTimeout);
TON7(IN:=(EXTRACT(X:=UBRAIN1.bButtons, N:=6) AND UBRAIN1.xValidRead), PT:=tTimeout);
TON8(IN:=(EXTRACT(X:=UBRAIN1.bButtons, N:=7) AND UBRAIN1.xValidRead), PT:=tTimeout*2);

TON10(IN:=(EXTRACT(X:=UBRAIN1.bDin1, N:=6) AND UBRAIN1.xValidRead), PT:=tTimeout);

resetAll := TON1.Q OR
			TON2.Q OR 
			TON3.Q OR 
			TON4.Q OR 
			TON5.Q OR 
			TON6.Q OR 
			TON7.Q OR 
			TON8.Q ;

Buttons[1]:=TON1.Q;
Buttons[2]:=TON2.Q;
Buttons[3]:=TON3.Q;
Buttons[4]:=TON4.Q;
Buttons[5]:=TON5.Q;
Buttons[6]:=TON6.Q;
Buttons[7]:=TON7.Q;
Buttons[8]:=TON8.Q;
Buttons[10]:=TON10.Q;
sumButtons := 0;
FOR i:=1 TO 10 DO
	sumButtons := sumButtons + BOOL_TO_INT(Buttons[i]);
END_FOR
IF sumButtons > 1 THEN
	FOR i:=1 TO 10 DO
		Buttons[i] := FALSE;
	END_FOR
END_IF
//_activeButton := EnumButton.NONE;

// Videos
IF Buttons[1] THEN
	GVL.glFlagStartVideo[1] := TRUE;
END_IF
IF Buttons[2] THEN
	GVL.glFlagStartVideo[2] := TRUE;
END_IF
IF Buttons[3] THEN
	GVL.glFlagStartVideo[3] := TRUE;
END_IF
IF Buttons[4] THEN
	GVL.glFlagStartVideo[4] := TRUE;
END_IF
IF Buttons[5] THEN
	GVL.glFlagStartVideo[5] := TRUE;
END_IF
IF Buttons[6] THEN
	GVL.glFlagStartVideo[6] := TRUE;
END_IF
IF Buttons[7] THEN
	GVL.glFlagStartVideo[7] := TRUE;
END_IF

//end Videos
// в режиме ожидания
IF(PLC_PRG.post.InWaitModes())THEN
	_activeButton := 0;

	// подсветка заблокированных функций
//	FOR i := EnumButton.BTN_ACTIVECLEAN TO EnumButton.BTN_PAUSE DO
	FOR i := 1 TO 8 DO
		IF(NOT DataFromSpk.GetAllowedButton(INT_TO_BYTE(i)))THEN
			DeviceLamps.SetAlarmLamps(i);
		ELSE
			DeviceLamps.SetLamps(i, FALSE);
		END_IF
	END_FOR;

//	FOR i := EnumButton.BTN_ACTIVECLEAN TO EnumButton.BTN_PAUSE DO
//		DeviceLamps.SetLamps(i, FALSE);
//	END_FOR;
END_IF

// работа в режиме мойки
IF(PLC_PRG.post.InPaidWashMode())THEN
	// подсветка заблокированных функций
//	FOR i := EnumButton.BTN_ACTIVECLEAN TO EnumButton.BTN_PAUSE DO
	FOR i := 1 TO 10 DO
		IF(i < 9)THEN	// исключая кнопку СТОП
			IF(NOT DataFromSpk.GetAllowedButton(INT_TO_BYTE(i)))THEN
				DeviceLamps.SetAlarmLamps(i);
			ELSE
				IF(i <> _activeButton AND NOT (i = EnumButton.BTN_COLDWATER AND _activeButton = EnumButton.BTN_HIGHPRESSURE))THEN
					DeviceLamps.SetLamps(i, FALSE);
				END_IF
			END_IF
		ELSIF(i = 10)THEN
			IF(NOT DataFromSpk.GetAllowedButton(INT_TO_BYTE(i)))THEN
				//DeviceLamps.SetAlarmLamps(i);
			ELSE
				IF(i <> _activeButton)THEN
					DeviceLamps.SetLamps(i, FALSE);
				END_IF
			END_IF
		END_IF
	END_FOR;

//	FOR i := EnumButton.BTN_ACTIVECLEAN TO EnumButton.BTN_PAUSE DO
	FOR i := 1 TO 10 DO
		IF(i < 9)THEN	// исключая кнопку СТОП
			IF(Buttons[i] AND DataFromSpk.GetAllowedButton(INT_TO_BYTE(i)))THEN
				// включать функции только при положительном балансе
				IF(PLC_PRG.post.CounterFund > 0)THEN
					_activeButton := i;
				END_IF
				
				Buttons[i] := FALSE;
				
				EXIT;	// break
			END_IF
		ELSE
			IF(i = 10 AND Buttons[i] AND DataFromSpk.GetAllowedButton(INT_TO_BYTE(14)))THEN
				// включать функции только при положительном балансе
				IF(PLC_PRG.post.CounterFund > 0)THEN
					_activeButton := i;
				END_IF
				
				Buttons[i] := FALSE;
				
				EXIT;	// break
			END_IF
		END_IF
	END_FOR;
END_IF;

// работа в режиме уборки
IF(PLC_PRG.post.InClearWashMode())THEN
	// подсветить недоступные оператору функции заблокированным
//	FOR i := EnumButton.BTN_ACTIVECLEAN TO EnumButton.BTN_PAUSE DO
	FOR i := 1 TO 8 DO
//		IF(i <> EnumButton.BTN_COLDWATER AND i <> EnumButton.BTN_HOTWATER AND i <> EnumButton.BTN_ACTIVECLEAN)THEN
		IF(i <> EnumButton.BTN_COLDWATER AND i <> EnumButton.BTN_HOTWATER)THEN
			DeviceLamps.SetAlarmLamps(i);
		END_IF
	END_FOR;

	// доступные оператору кнопки
	// кнопка "Холодная вода"
	i := EnumButton.BTN_COLDWATER;
	// включить подсветку
	IF(NOT DataFromSpk.GetAllowedButton(INT_TO_BYTE(i)))THEN
		DeviceLamps.SetAlarmLamps(i);
	ELSE
		IF(i <> _activeButton)THEN
			DeviceLamps.SetLamps(i, FALSE);
		END_IF
	END_IF
	// проверить нажатие
	IF(Buttons[i] AND DataFromSpk.GetAllowedButton(INT_TO_BYTE(i)))THEN
		// включать функции только при уборке
		IF(NOT PLC_PRG.post.ModePaid)THEN
			_activeButton := i;
		END_IF
			
		Buttons[i] := FALSE;
	END_IF

	// кнопка "Горячая вода"
	i := EnumButton.BTN_HOTWATER;
	// включить подсветку
	IF(NOT DataFromSpk.GetAllowedButton(INT_TO_BYTE(i)))THEN
		DeviceLamps.SetAlarmLamps(i);
	ELSE
		IF(i <> _activeButton)THEN
			DeviceLamps.SetLamps(i, FALSE);
		END_IF
	END_IF
	// проверить нажатие
	IF(Buttons[i] AND DataFromSpk.GetAllowedButton(INT_TO_BYTE(i)))THEN
		// включать функции только при уборке
		IF(NOT PLC_PRG.post.ModePaid)THEN
			_activeButton := i;
		END_IF
			
		Buttons[i] := FALSE;
	END_IF
(*
	// кнопка "Активная химия" - открыть верхний замок
	i := EnumButton.BTN_ACTIVECLEAN;
	// включить подсветку
	IF(NOT PLC_PRG.post.IsUnlocked(EnumLock.LOCK_TOP)) THEN
		DeviceLamps.SetLampColor(i, DeviceLamps.COLOR_YELLOW);
	ELSE
		DeviceLamps.SetLampColor(i, DeviceLamps.COLOR_GREEN);
	END_IF
	// проверить нажатие
	IF(Buttons[i])THEN
		IF(NOT PLC_PRG.post.IsUnlocked(EnumLock.LOCK_TOP))THEN
			PLC_PRG.post.UnLock(EnumLock.LOCK_TOP, TRUE);	
		END_IF
			
		Buttons[i] := FALSE;
	END_IF
*)
END_IF;

// работа в режиме инкассации
IF(PLC_PRG.post.Mode = EnumMode.CASHCOLLECT)THEN
	btnStartEnable := EnumButton.BTN_SHAMPOO;
	btnStopEnable := EnumButton.BTN_FOAM;
	
	_activeButton := 0;
	FOR i := EnumButton.BTN_ACTIVECLEAN TO EnumButton.BTN_PAUSE DO
		IF(i <> EnumButton.BTN_SHAMPOO AND i <> EnumButton.BTN_ACTIVECLEAN AND i <> EnumButton.BTN_FOAM)THEN
			DeviceLamps.SetLamps(i, FALSE);
		END_IF
	END_FOR;
	
	IF(PLC_PRG.post.Locks[EnumLock.LOCK_TOP])THEN	
//		IF(NOT PLC_PRG.post.IsUnlocked(EnumLock.LOCK_TOP)) THEN
			DeviceLamps.SetLampColor(EnumButton.BTN_SHAMPOO, DeviceLamps.COLOR_YELLOW);
			DeviceLamps.SetLampColor(EnumButton.BTN_FOAM, DeviceLamps.COLOR_WHITE);
//		ELSE
//			DeviceLamps.SetLampColor(EnumButton.BTN_SHAMPOO, DeviceLamps.COLOR_WHITE);
//			DeviceLamps.SetLampColor(EnumButton.BTN_FOAM, DeviceLamps.COLOR_YELLOW);
//		END_IF
		
//		DeviceLamps.SetLamps(EnumButton.BTN_COLDWATER, FALSE);
	ELSE
//		DeviceLamps.SetLamps(EnumButton.BTN_COLDWATER, TRUE);	
			DeviceLamps.SetLampColor(EnumButton.BTN_SHAMPOO, DeviceLamps.COLOR_WHITE);
			DeviceLamps.SetLampColor(EnumButton.BTN_FOAM, DeviceLamps.COLOR_YELLOW);
	END_IF
	
//	IF(PLC_PRG.post.Locks[EnumLock.LOCK_MID])THEN
//		IF(NOT PLC_PRG.post.IsUnlocked(EnumLock.LOCK_MID)) THEN
//			DeviceLamps.SetLampColor(EnumButton.BTN_FOAM, DeviceLamps.COLOR_YELLOW);
//		ELSE
//			DeviceLamps.SetLampColor(EnumButton.BTN_FOAM, DeviceLamps.COLOR_GREEN);
//		END_IF
//		
////		DeviceLamps.SetLamps(EnumButton.BTN_HOTWATER, FALSE);
//	ELSE
////		DeviceLamps.SetLamps(EnumButton.BTN_HOTWATER, TRUE);	
//	END_IF
	
//	// кнопка инкассации доступна после открытия обеих дверей
//	IF(NOT PLC_PRG.post.Locks[EnumLock.LOCK_TOP] AND NOT PLC_PRG.post.Locks[EnumLock.LOCK_MID])THEN
	// кнопка инкассации доступна после открытия ОДНОЙ дверей
	IF(NOT PLC_PRG.post.Locks[EnumLock.LOCK_TOP])THEN
		IF(NOT fBtnCollectPushed)THEN
			DeviceLamps.SetLampColor(EnumButton.BTN_ACTIVECLEAN, DeviceLamps.COLOR_GREEN);
		ELSE
			DeviceLamps.SetLampColor(EnumButton.BTN_ACTIVECLEAN, DeviceLamps.COLOR_BLUE);
		END_IF
		
//		// разрешать нажимать инкассацию после открытия обеих дверей
//		btnStopEnable := EnumButton.BTN_FOAM;
//	ELSE
//		DeviceLamps.SetLampColor(EnumButton.BTN_FOAM, DeviceLamps.COLOR_WHITE);
//		
//		btnStopEnable := EnumButton.BTN_FOAM;
	END_IF

	FOR i := btnStartEnable TO btnStopEnable DO
		IF(Buttons[i])THEN
			_activeButton := i;
			
			Buttons[i] := FALSE;
			
			EXIT;	// break
		END_IF;
	END_FOR;

	// установить факт нажатия кнопки инкассации
	IF(_activeButton = EnumButton.BTN_ACTIVECLEAN)THEN
		// допускать только одно нажатие кнопки инкассации
		IF(fBtnCollectPushed)THEN
			_activeButton := 0;
		END_IF
		
		fBtnCollectPushed := TRUE;
	END_IF
END_IF;

// работа в режиме сервиса
IF(PLC_PRG.post.InServiceMode())THEN
	// подсветка заблокированных функций
	//FOR i := EnumButton.BTN_ACTIVECLEAN TO EnumButton.BTN_PAUSE DO
	FOR i := 1 TO 8 DO
		IF(NOT DataFromSpk.GetAllowedButton(INT_TO_BYTE(i)))THEN
			DeviceLamps.SetAlarmLamps(i);
		ELSE
			IF(i <> _activeButton)THEN
				DeviceLamps.SetLamps(i, FALSE);
			END_IF
		END_IF
	END_FOR;

	//FOR i := EnumButton.BTN_ACTIVECLEAN TO EnumButton.BTN_PAUSE DO
	FOR i := 1 TO 8 DO
		IF(Buttons[i] AND DataFromSpk.GetAllowedButton(INT_TO_BYTE(i)))THEN
			// включать функции только при положительном балансе
			IF(NOT PLC_PRG.post.ModePaid)THEN
				_activeButton := i;
			END_IF
			
			Buttons[i] := FALSE;
			
			EXIT;	// break
		END_IF
	END_FOR;
END_IF;

// работа в режиме добавления денег
IF(PLC_PRG.post.Mode = EnumMode.FREEMONEY)THEN
	_activeButton := 0;
//	FOR i := EnumButton.BTN_ACTIVECLEAN TO EnumButton.BTN_PAUSE DO
	FOR i := 1 TO 8 DO
		DeviceLamps.SetLamps(i, FALSE);
	END_FOR;
	
	DeviceLamps.SetLamps(EnumButton.BTN_ACTIVECLEAN, TRUE);
	DeviceLamps.SetLamps(EnumButton.BTN_FOAM, TRUE);

//	FOR i := EnumButton.BTN_ACTIVECLEAN TO EnumButton.BTN_PAUSE DO
	FOR i := 1 TO 8 DO
		IF(Buttons[i])THEN
			_activeButton := i;
			
			Buttons[i] := FALSE;
			
			EXIT;	// break
		END_IF;
	END_FOR;
END_IF;


// Проверить нажатие кнопки завершения
Buttons[9] := EXTRACT(X:=UBRAIN1.bDin1, N:=3) AND UBRAIN1.xValidRead;
IF(Buttons[9] AND (PLC_PRG.post.ActiveCardType <> EnumCardType.UNDEFINED)) THEN
	PLC_PRG.post.OnFinButton();	

	//DeviceOut.SetOut(DeviceOut.OUT_COLOR_BTN_STOP, TRUE);
	
	//DeviceOut.SetOut(OUT_COLOR_BTN_STOP, TRUE);
	//TP9(IN:= FALSE, PT:= T#1S);
	
	TP9(IN:= TRUE, PT:= T#1S);
END_IF
TP9(in:=FALSE);
DeviceOut.SetOut(DeviceOut.OUT_COLOR_BTN_STOP_BIT, TP9.Q);

// после нажатия кнопки завершения сбрасывать кнопку активной функции
IF(Buttons[9])THEN
	// сбрасывать текущую кнопку только не для режима мойки
	IF(NOT PLC_PRG.post.InPaidWashMode())THEN
		_activeButton := EnumButton.NONE;
	END_IF
	
	// помечать замки закрытыми
	PLC_PRG.post.UnLock(EnumLock.LOCK_TOP, FALSE);
	PLC_PRG.post.UnLock(EnumLock.LOCK_MID, FALSE);
	
	// сбросить факт нажатия кнопки инкассации
	fBtnCollectPushed := FALSE;
	
	// печатать чек
	IF(PLC_PRG.post.lastInCash > 0)THEN
		SysTimeRtcConvertUtcToLocal(SysTimeRtcGet(udiResult), udiTimeLocal);
		timeDate:= UDINT_TO_DT(udiTimeLocal);
		DevicePrinter.PrintBill(printingTime := OSCAT_BASIC.UTC_TO_LTIME(timeDate, DST_ENABLE :=0, TIME_ZONE_OFFSET:=DevicePrinter.TIME_ZONE_MINUTES_OFFSET), costWash := PLC_PRG.post.lastInCash);
		
		PLC_PRG.post.SetLastInCash(0);
	END_IF
END_IF

//IF(_activeButton <> externalActiveButton AND externalActiveButton = EnumButton.NONE)THEN
IF(_activeButton <> externalActiveButton)THEN
	// погасить лампу текущего режима
	DeviceLamps.SetLamps(externalActiveButton, FALSE);
	// для ТурбоСмыва одновременно зажигать кнопку ХВ
	IF(externalActiveButton = EnumButton.BTN_HIGHPRESSURE)THEN
		DeviceLamps.SetLamps(EnumButton.BTN_COLDWATER, FALSE);
	END_IF
	
	//IF(PLC_PRG.post.Mode <> EnumMode.CASHCOLLECT)THEN
		externalActiveButton := _activeButton;
	//END_IF

	// включить лампу нового режима
	IF(PLC_PRG.post.CounterFund > 0 OR NOT PLC_PRG.post.ModePaid)THEN
		DeviceLamps.SetLamps(externalActiveButton, TRUE);
		// для ТурбоСмыва одновременно зажигать кнопку ХВ
		IF(externalActiveButton = EnumButton.BTN_HIGHPRESSURE)THEN
			DeviceLamps.SetLamps(EnumButton.BTN_COLDWATER, TRUE);
		END_IF
	END_IF
END_IF

//// Проверить нажатие кнопки ХВ высокого давления
////Buttons[10] := EXTRACT(X:=UBRAIN1.bDin1, N:=6) AND UBRAIN1.xValidRead;
//IF( Buttons[10] ) THEN
//	
//	IF SPK_DATA.go_postNumber > 0 THEN
//		SPK_DATA.go_postNumber := 0;
//		DeviceLamps.SetLightTurbo(FALSE);
////		DeviceLamps.SetIllumination(DeviceLamps.ILLUMINATION_COLOR_RED);
//	ELSE
//		SPK_DATA.go_postNumber := 1;	
//		DeviceLamps.SetLightTurbo(TRUE);
////		DeviceLamps.SetIllumination(DeviceLamps.ILLUMINATION_COLOR_YELLOW);
//	END_IF
//	// переключить TURBO
//	//PLC_PRG.post.OnFinButton();	
//
//	//DeviceOut.SetOut(DeviceOut.OUT_COLOR_BTN_STOP, TRUE);
//	
//	//DeviceOut.SetOut(OUT_COLOR_BTN_STOP, TRUE);
//	//TP9(IN:= FALSE, PT:= T#1S);
//	
////	TP10(IN:= TRUE, PT:= T#1S);
//END_IF
//TP10(in:=FALSE);
//DeviceOut.SetOut(DeviceOut.OUT_COLOR_BTN_STOP_BIT, TP9.Q);

METHOD PUBLIC GetActiveButton : int
VAR_INPUT
END_VAR
GetActiveButton := externalActiveButton;

// кнопка ХВ высокого давления
IF(externalActiveButton = 10)THEN
	GetActiveButton := 14;
END_IF

IF(GetActiveButton = 1)THEN
	GetActiveButton := 2;
ELSIF(GetActiveButton = 2)THEN
	GetActiveButton := 1;
END_IF

//externalActiveButton := EnumButton.NONE;
END_METHOD

END_PROGRAM

// CompWin/AppTerminalPost/Traffic/DataFromSpk
PROGRAM DataFromSpk
VAR
//	r_trig_XXX : R_TRIG;
//	tp_XXX : TP;
//	kk : INT;
	
	needNewTarif : BOOL := FALSE;
	i : BYTE;

	needNewPause : BOOL := FALSE;
END_VAR

// ВНИМАНИЕ! цена gi_rates[8] не приходит от DataFromSpk
// новые тарифы
IF(SPK_DATA.gi_rateSave = 1 AND PLC_PRG.post.InWaitModes())THEN
	needNewTarif := FALSE;
	FOR i := 0 TO 8 DO
		IF(PersistentVars.rates[i] <> SPK_DATA.gi_rates[i])THEN
			needNewTarif := TRUE;
			EXIT;	// break
		END_IF
	END_FOR
	
	IF(needNewTarif)THEN
		PLC_PRG.post.SaveNewRates();
	END_IF
END_IF

// новые паузы
IF(SPK_DATA.gi_pauseSave = 1 AND PLC_PRG.post.InWaitModes())THEN
	needNewPause := FALSE;
	
	IF(NOT needNewPause AND (PLC_PRG.post.GetPauseActiveClean() <> WORD_TO_TIME(1000 * SPK_DATA.gi_pauseActiveClean)))THEN
		needNewPause := TRUE;
	END_IF
	
	IF(NOT needNewPause AND (PLC_PRG.post.GetPauseFoam() <> WORD_TO_TIME(1000 * SPK_DATA.gi_pauseFoam)))THEN
		needNewPause := TRUE;
	END_IF
	
	IF(NOT needNewPause AND (PLC_PRG.post.GetPauseShampoo() <> WORD_TO_TIME(1000 * SPK_DATA.gi_pauseShampoo)))THEN
		needNewPause := TRUE;
	END_IF
	
	IF(needNewPause)THEN
		PLC_PRG.post.SaveNewPause();
	END_IF
END_IF

(*
// при необходимости применить новые тарифы от сервера
r_trig_XXX(CLK:=WORD_TO_BOOL(SPK_DATA.gi_rateSave));

tp_XXX(IN := r_trig_XXX.Q, PT := T#2S);

IF(tp_XXX.Q)THEN
	needNewTarif := TRUE;
END_IF

IF(( needNewTarif ) AND PLC_PRG.post.InWaitModes())THEN
	PLC_PRG.post.SaveNewRates();
	// сбросить признак необходимости применения тарифов
	//SPK_DATA.gi_rateSave := 0;
	//kk := 8;
	
	needNewTarif := FALSE;
END_IF
*)

METHOD GetConfirmedMode : INT
VAR_INPUT
END_VAR
GetConfirmedMode := 0;

CASE SPK_DATA.gi_nCurFunction OF
	1:
		GetConfirmedMode := EnumMode.ACTIVECLEAN;
	2:
		GetConfirmedMode := EnumMode.FOAM;
	3:
		GetConfirmedMode := EnumMode.SHAMPOO;
	4:
		GetConfirmedMode := EnumMode.COLDWATER;
	5:
		GetConfirmedMode := EnumMode.HOTWATER;
	6:
		GetConfirmedMode := EnumMode.WAX;
	7:
		GetConfirmedMode := EnumMode.OSMOSE;
	8:
		GetConfirmedMode := EnumMode.PAUSE;
	14:
		GetConfirmedMode := EnumMode.HIGHPRESSURE;
		
		
END_CASE
END_METHOD

METHOD GetAllowedButton : BOOL
VAR_INPUT
	button: BYTE;
END_VAR

VAR
	i : BYTE;
	testFlag : BYTE;
END_VAR
GetAllowedButton := TRUE;

// замена для предварительной, интенсивной, пены и высокого давления
IF(button = 1)THEN
	testFlag := 2;
ELSIF(button = 2)THEN
	testFlag := 0;
ELSIF(button = 3)THEN
	testFlag := 1;
ELSIF(button = 14)THEN
	testFlag := 3;
ELSE
	testFlag := button - 1;	
END_IF

IF(testFlag <> 0)THEN
	GetAllowedButton := SPK_DATA.gi_aAllowedFlags[testFlag];
ELSE
	GetAllowedButton := FALSE;
	
	FOR i := 0 TO 7 DO
		IF(SPK_DATA.gi_aAllowedFlags[i])THEN
			GetAllowedButton := TRUE;
			EXIT;
		END_IF
	END_FOR
END_IF
END_METHOD

METHOD GetBonusValue : WORD
GetBonusValue := SPK_DATA.gi_bonusValue;
END_METHOD

METHOD GetAllowedMode : BOOL
VAR_INPUT
	mode: BYTE;
END_VAR

VAR
	i : BYTE;
	testFlag : BYTE;
END_VAR
GetAllowedMode := TRUE;

// замена для предварительной, интенсивной, пены и высокого давления
IF(mode = 1)THEN
	testFlag := 0;
ELSIF(mode = 2)THEN
	testFlag := 1;
ELSIF(mode = 3)THEN
	testFlag := 2;
ELSIF(mode = 14)THEN
	testFlag := 3;
ELSE
	testFlag := mode - 1;	
END_IF

IF(testFlag <> 0)THEN
	GetAllowedMode := SPK_DATA.gi_aAllowedFlags[testFlag];
ELSE
	GetAllowedMode := FALSE;
	
	FOR i := 0 TO 7 DO
		IF(SPK_DATA.gi_aAllowedFlags[i])THEN
			GetAllowedMode := TRUE;
			EXIT;
		END_IF
	END_FOR
END_IF
END_METHOD

END_PROGRAM

// CompWin/AppTerminalPost/DevOut/DeviceOut
// дискретные выхода поста
PROGRAM DeviceOut
VAR CONSTANT
	IN_DCOK_BIT :BYTE := 7;	//2#1000_0000;	// вход DCOK
	IN_TURBO_BUTTON_BIT :BYTE := 6;	//2#1000_0000;	// вход TURBO кнопки

	//OUT_ILLUMINATION: byte
	OUT_RELAY_BIT :BYTE := 0;	//2#0000_0001;	// выход реле
	
	OUT_COLOR_BTN_STOP_BIT : BYTE := 4;	//2#0001_0000;	// выход подсветки кнопки "Завершить"
	OUT_COLOR_BTN_HELP_BIT : BYTE := 5; //2#0010_0000;	// выход подсветки кнопки "Помощь"
	OUT_LOCK_TOP_BIT : BYTE := 6;	//2#0100_0000;			// верхний замок
	OUT_LOCK_MID_BIT : BYTE := 7;	//2#1000_0000;			// средний замок
END_VAR

VAR
	bDOut1 : BYTE := 0;
	
	TP_LOCK_TOP : TP;
	TP_LOCK_MID : TP;
	TP_SAVE_RETAIN : TP;
	//Outs : ARRAY [1 .. 2] OF BOOL := [FALSE];
	
	// Флаг наличия электропитания DC OK
	fDcOk : BOOL;
	TpDcOk : TOF;
	
	fShutdown : BOOL := FALSE;
END_VAR

// подключить аккумулятор
IF(NOT fShutdown)THEN
	DeviceOut.SetOut(DeviceOut.OUT_RELAY_BIT, TRUE);
END_IF

// Проверить DC OK
fDcOk := EXTRACT(X:=UBRAIN1.bDin1, N:= IN_DCOK_BIT)  AND UBRAIN1.xValidRead;
//TpDcOk(IN:= fDcOk, PT:= T#5S);
// Контролировать связь с UBrain
TpDcOk(IN:= fDcOk AND UBRAIN1.xValidRead AND UBRAIN1.xValidWrite, PT:= T#5S);
(*
IF(NOT fDcOk)THEN
	// взвести таймер отключения
	TpDcOk(IN:= TRUE, PT:= T#10S);
END_IF

TpDcOk();
*)
// если прошло время, а питание не появилось, то отключить контроллер
TpDcOk();
IF(NOT TpDcOk.Q AND NOT PLC_PRG.appStatus.startFlag)THEN
	// пропало электропитание
	PLC_PRG.post.OnLowPower();
	
	//// выставить флаг необходимости считывания retain переменных из файла
	//PLC_PRG.appStatus.startFlag := TRUE;
	
	
	TP_SAVE_RETAIN(IN:=TRUE, pt:=T#10S);
	TP_SAVE_RETAIN(IN:=FALSE);
	// выключить контроллер
	IF ( NOT TP_SAVE_RETAIN.Q) THEN
		PLC_PRG.post.Shutdown();
		fShutdown := TRUE; 
	END_IF;
ELSE
	fShutdown := FALSE;
END_IF


// верхний замок
//IF(((UBRAIN1.bDOut1 AND 2#0100_0000) <> 0)) THEN
IF(PLC_PRG.post.IsUnlocked(EnumLock.LOCK_TOP)) THEN
	TP_LOCK_TOP(IN:= TRUE, PT:= T#500MS);
END_IF
TP_LOCK_TOP(in:=FALSE);
DeviceOut.SetOut(DeviceOut.OUT_LOCK_TOP_BIT, (TP_LOCK_TOP.Q AND NOT TP_LOCK_MID.Q) );

// средний замок
//IF(((UBRAIN1.bDOut1 AND 2#1000_0000) <> 0))THEN
IF(PLC_PRG.post.IsUnlocked(EnumLock.LOCK_MID)) THEN
	TP_LOCK_MID(IN:= TRUE, PT:= T#500MS);
END_IF
TP_LOCK_MID(in:=FALSE);
DeviceOut.SetOut(DeviceOut.OUT_LOCK_MID_BIT, (TP_LOCK_MID.Q AND NOT TP_LOCK_TOP.Q) );

METHOD PUBLIC SetOut : INT
VAR_INPUT
	Idx0: BYTE;
	On: BOOL;
END_VAR
//Outs[Index] := On;

bDOut1 := UBRAIN1.bDOut1;
bDOut1 := DWORD_TO_BYTE(PUTBIT(bDOut1, Idx0, On));
	
UBRAIN1.bDOut1 := bDOut1;

SetOut := Idx0;
END_METHOD

END_PROGRAM

// CompWin/AppTerminalPost/DevPrinter/DevicePrinter
PROGRAM DevicePrinter
VAR CONSTANT
	PRINTER_FILE: CAA.FILENAME := '/dev/usb/lp0';
	TIME_ZONE_MINUTES_OFFSET : INT :=3*60;
END_VAR
VAR
	printer: printReceipt;
	receipt: receiptBuffer;
	i: INT;
	
	printFlag : BOOL := FALSE;
	
	timeDate: DATE_AND_TIME;
	
	udiResult: UDINT;
	udiTimeLocal : UDINT;
	
	xBusy : BOOL := FALSE;
END_VAR

IF printFlag THEN 
	IF printer.xExecute THEN
		printer(xExecute:=TRUE);
	ELSE
		xBusy := TRUE;
		printer(xExecute:=TRUE, printerFile:=PRINTER_FILE, receiptData:=ADR(receipt.buffer), receiptDataSize:=receipt.size);
	END_IF	

	IF printer.xDone OR printer.xError THEN
		xBusy := FALSE;
		printFlag := FALSE;
	END_IF
END_IF

METHOD printEncashment
VAR_INPUT
	printingTime : DATE_AND_TIME;
	
	countBanknote10 : WORD;
	countBanknote50 : WORD;
	countBanknote100 : WORD;
	
	countCoin10 : WORD;
	
	
END_VAR

VAR
//	// адрес мойки
//	washAddress : WSTRING :="Волгоград Жукова 55";
END_VAR
	receipt.clear();
	
	//init commands
	receipt.ejectTicket();
	receipt.initPrinter();
	receipt.setCP866Encoding();
	receipt.newline();
	//receipt template
	receipt.setFont(FONT_A);
	receipt.setFontBold(bold:=TRUE);
	receipt.setFontSize2(width:=1, height :=1);
	receipt.setFontAlignment(alignment := ALIGN_CENTER);
	receipt.println(PersistentVars.washAddress);
//	receipt.println(washAddress);
	receipt.newline();
	
	//DT_TO_STRF()
	receipt.setFont(FONT_B);
	receipt.setFontBold(bold:=TRUE);
	receipt.setFontSize2(width:=3, height :=3);
	receipt.setFontAlignment(alignment := ALIGN_CENTER);
	receipt.println("Инкассация");
	
	receipt.setFont(FONT_A);
	receipt.setFontSize2(width:=1, height :=1);
	receipt.setFontBold(bold:=FALSE);
	receipt.println(STRING_TO_WSTRING(OSCAT_BASIC.DT_TO_STRF(DTI:=printingTime,MS:=0, FMT:=WSTRING_TO_STRING("#N:#R #G.#C.#A"), LANG:=0)));
	receipt.newline();
	
	
	receipt.setFontBold(bold:=TRUE);
	receipt.setFontSize2(width:=2, height :=2);
	receipt.println(WCONCAT("Пост ", INT_TO_WSTRING(PLC_PRG.post.Number) ));
//	receipt.println(WCONCAT("Пост ", UINT_TO_WSTRING(postNumber) ));
	
	receipt.setFontAlignment(alignment := ALIGN_CENTER);
	receipt.setFontSize2(width:=1, height :=1);
	receipt.setFontBold(bold:=FALSE);
	
	
	receipt.println(WCONCAT("Количество банкнот 10р: ", WORD_TO_WSTRING(countBanknote10)));
	receipt.println(WCONCAT("Количество банкнот 50р: ", WORD_TO_WSTRING(countBanknote50)));
	receipt.println(WCONCAT("Количество банкнот 100р: ", WORD_TO_WSTRING(countBanknote100)));
	receipt.newline();
	receipt.println(WCONCAT("Количество монет 10р: ", WORD_TO_WSTRING(countCoin10)));
	receipt.newline();
	
//	IF banknoteCount > 0 THEN
//		receipt.println(WCONCAT("Количество банкнот ", UINT_TO_WSTRING(banknoteCount)));
//	END_IF
	
//	IF coinCount > 0 THEN
//		receipt.println(WCONCAT("Количество монет ", UINT_TO_WSTRING(coinCount)));
//	END_IF
	
	//receipt.setFont(FONT_B);
	//receipt.println("Итог");
	receipt.totalCut();
	receipt.presentPageAndTimeoutRetract(10); //show ticket and wait
	
	printFlag := TRUE;
END_METHOD

METHOD PrintBill
VAR_INPUT
	printingTime : DATE_AND_TIME;
	
	costWash : REAL;	
END_VAR

VAR
	wstr : WSTRING;
	cost : INT;
END_VAR
	receipt.clear();
	
	//init commands
	receipt.ejectTicket();
	receipt.initPrinter();
	receipt.setCP866Encoding();
	receipt.newline();
	//receipt template
	receipt.setFont(FONT_A);
	receipt.setFontBold(bold:=TRUE);
	receipt.setFontSize2(width:=1, height :=1);
	receipt.setFontAlignment(alignment := ALIGN_CENTER);
	receipt.println(PersistentVars.washAddress);
//	receipt.println(washAddress);
	receipt.newline();
	
	//DT_TO_STRF()
	receipt.setFont(FONT_B);
	receipt.setFontBold(bold:=TRUE);
	receipt.setFontSize2(width:=3, height :=3);
	receipt.setFontAlignment(alignment := ALIGN_CENTER);
	receipt.println("Мойка");
	
	receipt.setFont(FONT_A);
	receipt.setFontSize2(width:=1, height :=1);
	receipt.setFontBold(bold:=FALSE);
	receipt.println(STRING_TO_WSTRING(OSCAT_BASIC.DT_TO_STRF(DTI:=printingTime,MS:=0, FMT:=WSTRING_TO_STRING("#N:#R #G.#C.#A"), LANG:=0)));
	receipt.newline();
	
	
	receipt.setFontBold(bold:=TRUE);
	receipt.setFontSize2(width:=2, height :=2);
	receipt.println(WCONCAT("Пост ", INT_TO_WSTRING(PLC_PRG.post.Number) ));
//	receipt.println(WCONCAT("Пост ", UINT_TO_WSTRING(postNumber) ));
	
	receipt.setFontAlignment(alignment := ALIGN_CENTER);
	receipt.setFontSize2(width:=1, height :=1);
	receipt.setFontBold(bold:=FALSE);
	
	receipt.newline();

	// Для REAL отбросываю дробную часть DINT_TO_INT(TRUNC(real));
	cost := DINT_TO_INT(TRUNC(costWash));
	// REAL_TO_WORD(real);	// округление до ближайшего целого
	wstr := WCONCAT("Стоимость: ", INT_TO_WSTRING(cost));
	wstr := WCONCAT(wstr, " р.");
	receipt.println(wstr);
	receipt.newline();
	
//	IF banknoteCount > 0 THEN
//		receipt.println(WCONCAT("Количество банкнот ", UINT_TO_WSTRING(banknoteCount)));
//	END_IF
	
//	IF coinCount > 0 THEN
//		receipt.println(WCONCAT("Количество монет ", UINT_TO_WSTRING(coinCount)));
//	END_IF
	
	//receipt.setFont(FONT_B);
	//receipt.println("Итог");
	receipt.totalCut();
	receipt.presentPageAndTimeoutRetract(10); //show ticket and wait
	
	printFlag := TRUE;
END_METHOD

END_PROGRAM

// CompWin/AppTerminalPost/DevPrinter/printReceipt
///command with  no-data ack
FUNCTION_BLOCK printReceipt
VAR CONSTANT
	STATE_INITIAL: BYTE := 0;
	STATE_WRITE: BYTE := 1;
	STATE_FATAL_ERROR: BYTE := 3;
	STATE_CLOSE: BYTE := 4;
END_VAR
VAR_INPUT
	xExecute: BOOL := FALSE;
	printerFile: STRING(255);
	receiptData: POINTER TO BYTE;
	receiptDataSize: CAA.SIZE := 0;
END_VAR
VAR
	///printerHandle :  RTS_IEC_HANDLE;
	printerOpen: File.Open;
	printerClose: File.Close;
	printerWrite: File.Write;
	state: BYTE := STATE_INITIAL;
	reenterStateMachine: BOOL;
END_VAR
VAR_OUTPUT
	xDone: BOOL := FALSE;
	xError: BOOL := FALSE;
	xBusy: BOOL := FALSE;
	xErrorCode: PRINTER_ERROR := PRINTER_NO_ERROR;
END_VAR

REPEAT
	reenterStateMachine := FALSE;
CASE state OF 
	STATE_INITIAL:
		IF xExecute THEN
			xDone := FALSE;
			xError := FALSE;
			xBusy := TRUE;
			printerOpen (xExecute := TRUE, sFileName := printerFile,
				eFileMode := FILE.MODE.MWRITE, xExclusive:= FALSE			
			);
			
			IF printerOpen.xDone THEN 
				xDone := FALSE;
				state := STATE_WRITE;
				reenterStateMachine := TRUE;
				printerWrite(xExecute:=FALSE);
				printerClose(xExecute:=FALSE);
			END_IF
			
			IF printerOpen.xError THEN 
				xError := TRUE;
				xExecute := FALSE;
				xBusy := FALSE;
				xErrorCode := PRINTER_FILE_OPEN_ERROR;
				state := STATE_INITIAL;
			END_IF
		
		END_IF
		//waiting ACK
	STATE_WRITE:
		printerWrite(xExecute :=TRUE, hFile := printerOpen.hFile, pBuffer := receiptData, szSize := receiptDataSize);
		IF printerWrite.xDone THEN
			state:=STATE_CLOSE;
			reenterStateMachine := TRUE;
		END_IF
		
		IF printerWrite.xError THEN
			state:= STATE_CLOSE;
			xError := TRUE;
			reenterStateMachine := TRUE;
			xErrorCode := PRINTER_WRITE_ERROR;
		END_IF
	STATE_CLOSE:
		state := STATE_INITIAL;
		IF printerOpen.xDone THEN
			xBusy := FALSE;
			xDone :=  NOT (xError);
			printerClose(hFile:=printerOpen.hFile);
		END_IF
		
END_CASE

UNTIL NOT (reenterStateMachine) 
END_REPEAT

END_FUNCTION_BLOCK

// CompWin/AppTerminalPost/DevPrinter/receiptBuffer
///буфер для формирования чека
FUNCTION_BLOCK receiptBuffer
VAR CONSTANT
	MAX_BUFFER_SIZE: UINT := 4096;
END_VAR
VAR
	size: UINT := 0;
	buffer: ARRAY[0..(MAX_BUFFER_SIZE - 1)] OF BYTE;
END_VAR

///set cpi (characters per inch). Working once (?)
METHOD setFontCPI
VAR
	SET_FONT_CPI_COMMAND: ARRAY[0..2] OF BYTE := [16#1B, 16#C1, 16#0];
END_VAR
VAR_INPUT
	printerCPI: PRINTER_FONT_CPI;
END_VAR

SET_FONT_CPI_COMMAND [2] := printerCPI;
push_back_array(xArray:=ADR(SET_FONT_CPI_COMMAND ), xArraySize:=UINT_TO_BYTE(SIZEOF(SET_FONT_CPI_COMMAND )));
END_METHOD

///set cpi (characters per inch). Working once (?)
METHOD setFontSize
VAR
	SET_FONT_SIZE_COMMAND: ARRAY[0..2] OF BYTE := [16#1B, 16#4D, 16#0];
END_VAR
VAR_INPUT
	printerFontSize: PRINTER_FONT_SIZE;
END_VAR

SET_FONT_SIZE_COMMAND[2] := printerFontSize;
push_back_array(xArray:=ADR(SET_FONT_SIZE_COMMAND), xArraySize:=UINT_TO_BYTE(SIZEOF(SET_FONT_SIZE_COMMAND)));
END_METHOD

METHOD clear
size:=0;
END_METHOD

///print unicode text
METHOD print
VAR_INPUT
	text: WSTRING(255);
END_VAR
VAR
	i: INT;
	char: UINT;
	cp866char: BYTE;
END_VAR
FOR i:=0 TO WLEN(text)-1 DO
	cp866char:= unicodeSymbol2cp866(text[i]);
	push_back(cp866char);
END_FOR
END_METHOD

METHOD push_back
VAR_INPUT
	char: BYTE;
END_VAR
buffer[size]:=char;
size:=size+1;
END_METHOD

METHOD newline
VAR CONSTANT
	LF: BYTE := 16#A;
END_VAR
push_back(LF);
END_METHOD

///append array to back of buffer
METHOD push_back_array
VAR_INPUT
	xArray: POINTER TO BYTE;
	xArraySize: BYTE := 0;
END_VAR
Mem.MemMove(xArray, ADR(buffer) + size, xArraySize);
size:=size + xArraySize;
END_METHOD

METHOD setCP866Encoding
VAR CONSTANT
	SELECT_CHARACTER_TABLE: ARRAY[0..2] OF BYTE := [16#1B, 16#74, 16#11];
END_VAR
push_back_array(xArray:=ADR(SELECT_CHARACTER_TABLE), xArraySize:=UINT_TO_BYTE(SIZEOF(SELECT_CHARACTER_TABLE )));
END_METHOD

METHOD totalCut
VAR CONSTANT
	TOTAL_CUT_COMMAND: ARRAY[0..1] OF BYTE := [16#1B, 16#69];
END_VAR
push_back_array(xArray:=ADR(TOTAL_CUT_COMMAND), xArraySize:=UINT_TO_BYTE(SIZEOF(TOTAL_CUT_COMMAND)));
END_METHOD

METHOD initPrinter
VAR CONSTANT
	INITPRINTER_COMMAND: ARRAY[0..1] OF BYTE := [16#1B, 16#40];
END_VAR
push_back_array(xArray:=ADR(INITPRINTER_COMMAND), xArraySize:=UINT_TO_BYTE(SIZEOF(INITPRINTER_COMMAND )));
END_METHOD

METHOD ejectTicket
VAR CONSTANT
	EJECT_TICKET_COMMAND: ARRAY[0..2] OF BYTE := [16#1D, 16#65, 16#5];
END_VAR
push_back_array(xArray:=ADR(EJECT_TICKET_COMMAND), xArraySize:=UINT_TO_BYTE(SIZEOF(EJECT_TICKET_COMMAND )));
END_METHOD

METHOD presentPageAndTimeoutRetract
VAR
	PRESENT_COMMAND: ARRAY[0..4] OF BYTE := [16#1D, 16#65, 16#20, 16#C, 16#5];
END_VAR
VAR_INPUT
	timeout: BYTE := 5;
END_VAR
PRESENT_COMMAND[4] := timeout;
push_back_array(xArray:=ADR(PRESENT_COMMAND), xArraySize:=UINT_TO_BYTE(SIZEOF(PRESENT_COMMAND)));
END_METHOD

METHOD setFontBold
VAR
	EMPHASIZED_COMMAND: ARRAY[0..2] OF BYTE := [16#1B, 16#45, 16#0];
END_VAR
VAR_INPUT
	bold: BOOL;
END_VAR
IF bold THEN
	EMPHASIZED_COMMAND[2] := 1;
ELSE
	EMPHASIZED_COMMAND[2] := 0;
END_IF
push_back_array(xArray:=ADR(EMPHASIZED_COMMAND), xArraySize:=UINT_TO_BYTE(SIZEOF(EMPHASIZED_COMMAND)));
END_METHOD

METHOD setFontAlignment
VAR
	ALIGNMENT_COMMAND: ARRAY[0..2] OF BYTE := [16#1B, 16#61, 16#0];
END_VAR
VAR_INPUT
	alignment: TEXT_ALIGNMENT;
END_VAR
ALIGNMENT_COMMAND[2] := alignment;
push_back_array(xArray:=ADR(ALIGNMENT_COMMAND), xArraySize:=UINT_TO_BYTE(SIZEOF(ALIGNMENT_COMMAND)));
END_METHOD

///print unicode text
METHOD println
VAR_INPUT
	text: WSTRING(255);
END_VAR
print(text);
newline();
END_METHOD

///print unicode text, adding spaces to fill desired length
METHOD printWithLeftPadding
VAR_INPUT
	text: WSTRING(255);
	desiredLen: BYTE;
END_VAR
VAR
	i: INT;
END_VAR
IF desiredLen > WLEN(text) THEN
	FOR i:=0 TO desiredLen - WLEN(text) -1 DO
		push_back(16#20);
	END_FOR	
END_IF

print(text);
END_METHOD

///print unicode text into 2 columns, adding space to fill desired len
METHOD print2Colsln
VAR_INPUT
	leftText: WSTRING(255);
	rightText: WSTRING(255);
	desiredLen: BYTE;
END_VAR
VAR
	i: INT;
END_VAR
print(leftText);
IF desiredLen > (WLEN(leftText) + WLEN(rightText)) THEN
	FOR i:=0 TO desiredLen - WLEN(leftText) - WLEN(rightText) DO
		push_back(16#20);
	END_FOR	
END_IF

print(rightText);
newline();
END_METHOD

METHOD setFont
VAR
	SET_FONT_COMMAND: ARRAY[0..2] OF BYTE := [16#1B, 16#21, 16#0];
END_VAR
VAR_INPUT
	printerFont: PRINTER_FONT;
END_VAR

SET_FONT_COMMAND[2] := printerFont;
push_back_array(xArray:=ADR(SET_FONT_COMMAND), xArraySize:=UINT_TO_BYTE(SIZEOF(SET_FONT_COMMAND)));
END_METHOD

///set cpi (characters per inch). Working once (?)
METHOD setFontSize2
VAR
	SET_FONT_SIZE_COMMAND: ARRAY[0..2] OF BYTE := [16#1D, 16#21, 16#0];
END_VAR
VAR_INPUT
	///1 -normal, 2- 2x, 3-x.. 8-8x
	height: BYTE;
	///1 -normal, 2- 2x, 3-x.. 8-8x
	width: BYTE;
END_VAR

SET_FONT_SIZE_COMMAND[2] := (width-1) * 16 + (height -1) ;
push_back_array(xArray:=ADR(SET_FONT_SIZE_COMMAND), xArraySize:=UINT_TO_BYTE(SIZEOF(SET_FONT_SIZE_COMMAND)));
END_METHOD

END_FUNCTION_BLOCK

// CompWin/AppTerminalPost/DevPrinter/unicodeSymbol2cp866
///convert unicode symbol to unicodeSymbol2cp866 symbol
FUNCTION unicodeSymbol2cp866 : BYTE
VAR_INPUT
	charUnicode: UINT;
END_VAR

	CASE charUnicode OF
		16#0 : unicodeSymbol2cp866:=16#0;
		16#1 : unicodeSymbol2cp866:=16#1;
		16#2 : unicodeSymbol2cp866:=16#2;
		16#3 : unicodeSymbol2cp866:=16#3;
		16#4 : unicodeSymbol2cp866:=16#4;
		16#5 : unicodeSymbol2cp866:=16#5;
		16#6 : unicodeSymbol2cp866:=16#6;
		16#7 : unicodeSymbol2cp866:=16#7;
		16#8 : unicodeSymbol2cp866:=16#8;
		16#9 : unicodeSymbol2cp866:=16#9;
		16#A : unicodeSymbol2cp866:=16#A;
		16#B : unicodeSymbol2cp866:=16#B;
		16#C : unicodeSymbol2cp866:=16#C;
		16#D : unicodeSymbol2cp866:=16#D;
		16#E : unicodeSymbol2cp866:=16#E;
		16#F : unicodeSymbol2cp866:=16#F;
		16#10 : unicodeSymbol2cp866:=16#10;
		16#11 : unicodeSymbol2cp866:=16#11;
		16#12 : unicodeSymbol2cp866:=16#12;
		16#13 : unicodeSymbol2cp866:=16#13;
		16#14 : unicodeSymbol2cp866:=16#14;
		16#15 : unicodeSymbol2cp866:=16#15;
		16#16 : unicodeSymbol2cp866:=16#16;
		16#17 : unicodeSymbol2cp866:=16#17;
		16#18 : unicodeSymbol2cp866:=16#18;
		16#19 : unicodeSymbol2cp866:=16#19;
		16#1A : unicodeSymbol2cp866:=16#1A;
		16#1B : unicodeSymbol2cp866:=16#1B;
		16#1C : unicodeSymbol2cp866:=16#1C;
		16#1D : unicodeSymbol2cp866:=16#1D;
		16#1E : unicodeSymbol2cp866:=16#1E;
		16#1F : unicodeSymbol2cp866:=16#1F;
		16#20 : unicodeSymbol2cp866:=16#20;
		16#21 : unicodeSymbol2cp866:=16#21;
		16#22 : unicodeSymbol2cp866:=16#22;
		16#23 : unicodeSymbol2cp866:=16#23;
		16#24 : unicodeSymbol2cp866:=16#24;
		16#25 : unicodeSymbol2cp866:=16#25;
		16#26 : unicodeSymbol2cp866:=16#26;
		16#27 : unicodeSymbol2cp866:=16#27;
		16#28 : unicodeSymbol2cp866:=16#28;
		16#29 : unicodeSymbol2cp866:=16#29;
		16#2A : unicodeSymbol2cp866:=16#2A;
		16#2B : unicodeSymbol2cp866:=16#2B;
		16#2C : unicodeSymbol2cp866:=16#2C;
		16#2D : unicodeSymbol2cp866:=16#2D;
		16#2E : unicodeSymbol2cp866:=16#2E;
		16#2F : unicodeSymbol2cp866:=16#2F;
		16#30 : unicodeSymbol2cp866:=16#30;
		16#31 : unicodeSymbol2cp866:=16#31;
		16#32 : unicodeSymbol2cp866:=16#32;
		16#33 : unicodeSymbol2cp866:=16#33;
		16#34 : unicodeSymbol2cp866:=16#34;
		16#35 : unicodeSymbol2cp866:=16#35;
		16#36 : unicodeSymbol2cp866:=16#36;
		16#37 : unicodeSymbol2cp866:=16#37;
		16#38 : unicodeSymbol2cp866:=16#38;
		16#39 : unicodeSymbol2cp866:=16#39;
		16#3A : unicodeSymbol2cp866:=16#3A;
		16#3B : unicodeSymbol2cp866:=16#3B;
		16#3C : unicodeSymbol2cp866:=16#3C;
		16#3D : unicodeSymbol2cp866:=16#3D;
		16#3E : unicodeSymbol2cp866:=16#3E;
		16#3F : unicodeSymbol2cp866:=16#3F;
		16#40 : unicodeSymbol2cp866:=16#40;
		16#41 : unicodeSymbol2cp866:=16#41;
		16#42 : unicodeSymbol2cp866:=16#42;
		16#43 : unicodeSymbol2cp866:=16#43;
		16#44 : unicodeSymbol2cp866:=16#44;
		16#45 : unicodeSymbol2cp866:=16#45;
		16#46 : unicodeSymbol2cp866:=16#46;
		16#47 : unicodeSymbol2cp866:=16#47;
		16#48 : unicodeSymbol2cp866:=16#48;
		16#49 : unicodeSymbol2cp866:=16#49;
		16#4A : unicodeSymbol2cp866:=16#4A;
		16#4B : unicodeSymbol2cp866:=16#4B;
		16#4C : unicodeSymbol2cp866:=16#4C;
		16#4D : unicodeSymbol2cp866:=16#4D;
		16#4E : unicodeSymbol2cp866:=16#4E;
		16#4F : unicodeSymbol2cp866:=16#4F;
		16#50 : unicodeSymbol2cp866:=16#50;
		16#51 : unicodeSymbol2cp866:=16#51;
		16#52 : unicodeSymbol2cp866:=16#52;
		16#53 : unicodeSymbol2cp866:=16#53;
		16#54 : unicodeSymbol2cp866:=16#54;
		16#55 : unicodeSymbol2cp866:=16#55;
		16#56 : unicodeSymbol2cp866:=16#56;
		16#57 : unicodeSymbol2cp866:=16#57;
		16#58 : unicodeSymbol2cp866:=16#58;
		16#59 : unicodeSymbol2cp866:=16#59;
		16#5A : unicodeSymbol2cp866:=16#5A;
		16#5B : unicodeSymbol2cp866:=16#5B;
		16#5C : unicodeSymbol2cp866:=16#5C;
		16#5D : unicodeSymbol2cp866:=16#5D;
		16#5E : unicodeSymbol2cp866:=16#5E;
		16#5F : unicodeSymbol2cp866:=16#5F;
		16#60 : unicodeSymbol2cp866:=16#60;
		16#61 : unicodeSymbol2cp866:=16#61;
		16#62 : unicodeSymbol2cp866:=16#62;
		16#63 : unicodeSymbol2cp866:=16#63;
		16#64 : unicodeSymbol2cp866:=16#64;
		16#65 : unicodeSymbol2cp866:=16#65;
		16#66 : unicodeSymbol2cp866:=16#66;
		16#67 : unicodeSymbol2cp866:=16#67;
		16#68 : unicodeSymbol2cp866:=16#68;
		16#69 : unicodeSymbol2cp866:=16#69;
		16#6A : unicodeSymbol2cp866:=16#6A;
		16#6B : unicodeSymbol2cp866:=16#6B;
		16#6C : unicodeSymbol2cp866:=16#6C;
		16#6D : unicodeSymbol2cp866:=16#6D;
		16#6E : unicodeSymbol2cp866:=16#6E;
		16#6F : unicodeSymbol2cp866:=16#6F;
		16#70 : unicodeSymbol2cp866:=16#70;
		16#71 : unicodeSymbol2cp866:=16#71;
		16#72 : unicodeSymbol2cp866:=16#72;
		16#73 : unicodeSymbol2cp866:=16#73;
		16#74 : unicodeSymbol2cp866:=16#74;
		16#75 : unicodeSymbol2cp866:=16#75;
		16#76 : unicodeSymbol2cp866:=16#76;
		16#77 : unicodeSymbol2cp866:=16#77;
		16#78 : unicodeSymbol2cp866:=16#78;
		16#79 : unicodeSymbol2cp866:=16#79;
		16#7A : unicodeSymbol2cp866:=16#7A;
		16#7B : unicodeSymbol2cp866:=16#7B;
		16#7C : unicodeSymbol2cp866:=16#7C;
		16#7D : unicodeSymbol2cp866:=16#7D;
		16#7E : unicodeSymbol2cp866:=16#7E;
		16#7F : unicodeSymbol2cp866:=16#7F;
		16#410 : unicodeSymbol2cp866:=16#80;
		16#411 : unicodeSymbol2cp866:=16#81;
		16#412 : unicodeSymbol2cp866:=16#82;
		16#413 : unicodeSymbol2cp866:=16#83;
		16#414 : unicodeSymbol2cp866:=16#84;
		16#415 : unicodeSymbol2cp866:=16#85;
		16#416 : unicodeSymbol2cp866:=16#86;
		16#417 : unicodeSymbol2cp866:=16#87;
		16#418 : unicodeSymbol2cp866:=16#88;
		16#419 : unicodeSymbol2cp866:=16#89;
		16#41A : unicodeSymbol2cp866:=16#8A;
		16#41B : unicodeSymbol2cp866:=16#8B;
		16#41C : unicodeSymbol2cp866:=16#8C;
		16#41D : unicodeSymbol2cp866:=16#8D;
		16#41E : unicodeSymbol2cp866:=16#8E;
		16#41F : unicodeSymbol2cp866:=16#8F;
		16#420 : unicodeSymbol2cp866:=16#90;
		16#421 : unicodeSymbol2cp866:=16#91;
		16#422 : unicodeSymbol2cp866:=16#92;
		16#423 : unicodeSymbol2cp866:=16#93;
		16#424 : unicodeSymbol2cp866:=16#94;
		16#425 : unicodeSymbol2cp866:=16#95;
		16#426 : unicodeSymbol2cp866:=16#96;
		16#427 : unicodeSymbol2cp866:=16#97;
		16#428 : unicodeSymbol2cp866:=16#98;
		16#429 : unicodeSymbol2cp866:=16#99;
		16#42A : unicodeSymbol2cp866:=16#9A;
		16#42B : unicodeSymbol2cp866:=16#9B;
		16#42C : unicodeSymbol2cp866:=16#9C;
		16#42D : unicodeSymbol2cp866:=16#9D;
		16#42E : unicodeSymbol2cp866:=16#9E;
		16#42F : unicodeSymbol2cp866:=16#9F;
		16#430 : unicodeSymbol2cp866:=16#A0;
		16#431 : unicodeSymbol2cp866:=16#A1;
		16#432 : unicodeSymbol2cp866:=16#A2;
		16#433 : unicodeSymbol2cp866:=16#A3;
		16#434 : unicodeSymbol2cp866:=16#A4;
		16#435 : unicodeSymbol2cp866:=16#A5;
		16#436 : unicodeSymbol2cp866:=16#A6;
		16#437 : unicodeSymbol2cp866:=16#A7;
		16#438 : unicodeSymbol2cp866:=16#A8;
		16#439 : unicodeSymbol2cp866:=16#A9;
		16#43A : unicodeSymbol2cp866:=16#AA;
		16#43B : unicodeSymbol2cp866:=16#AB;
		16#43C : unicodeSymbol2cp866:=16#AC;
		16#43D : unicodeSymbol2cp866:=16#AD;
		16#43E : unicodeSymbol2cp866:=16#AE;
		16#43F : unicodeSymbol2cp866:=16#AF;
		16#2591 : unicodeSymbol2cp866:=16#B0;
		16#2592 : unicodeSymbol2cp866:=16#B1;
		16#2593 : unicodeSymbol2cp866:=16#B2;
		16#2502 : unicodeSymbol2cp866:=16#B3;
		16#2524 : unicodeSymbol2cp866:=16#B4;
		16#2561 : unicodeSymbol2cp866:=16#B5;
		16#2562 : unicodeSymbol2cp866:=16#B6;
		16#2556 : unicodeSymbol2cp866:=16#B7;
		16#2555 : unicodeSymbol2cp866:=16#B8;
		16#2563 : unicodeSymbol2cp866:=16#B9;
		16#2551 : unicodeSymbol2cp866:=16#BA;
		16#2557 : unicodeSymbol2cp866:=16#BB;
		16#255D : unicodeSymbol2cp866:=16#BC;
		16#255C : unicodeSymbol2cp866:=16#BD;
		16#255B : unicodeSymbol2cp866:=16#BE;
		16#2510 : unicodeSymbol2cp866:=16#BF;
		16#2514 : unicodeSymbol2cp866:=16#C0;
		16#2534 : unicodeSymbol2cp866:=16#C1;
		16#252C : unicodeSymbol2cp866:=16#C2;
		16#251C : unicodeSymbol2cp866:=16#C3;
		16#2500 : unicodeSymbol2cp866:=16#C4;
		16#253C : unicodeSymbol2cp866:=16#C5;
		16#255E : unicodeSymbol2cp866:=16#C6;
		16#255F : unicodeSymbol2cp866:=16#C7;
		16#255A : unicodeSymbol2cp866:=16#C8;
		16#2554 : unicodeSymbol2cp866:=16#C9;
		16#2569 : unicodeSymbol2cp866:=16#CA;
		16#2566 : unicodeSymbol2cp866:=16#CB;
		16#2560 : unicodeSymbol2cp866:=16#CC;
		16#2550 : unicodeSymbol2cp866:=16#CD;
		16#256C : unicodeSymbol2cp866:=16#CE;
		16#2567 : unicodeSymbol2cp866:=16#CF;
		16#2568 : unicodeSymbol2cp866:=16#D0;
		16#2564 : unicodeSymbol2cp866:=16#D1;
		16#2565 : unicodeSymbol2cp866:=16#D2;
		16#2559 : unicodeSymbol2cp866:=16#D3;
		16#2558 : unicodeSymbol2cp866:=16#D4;
		16#2552 : unicodeSymbol2cp866:=16#D5;
		16#2553 : unicodeSymbol2cp866:=16#D6;
		16#256B : unicodeSymbol2cp866:=16#D7;
		16#256A : unicodeSymbol2cp866:=16#D8;
		16#2518 : unicodeSymbol2cp866:=16#D9;
		16#250C : unicodeSymbol2cp866:=16#DA;
		16#2588 : unicodeSymbol2cp866:=16#DB;
		16#2584 : unicodeSymbol2cp866:=16#DC;
		16#258C : unicodeSymbol2cp866:=16#DD;
		16#2590 : unicodeSymbol2cp866:=16#DE;
		16#2580 : unicodeSymbol2cp866:=16#DF;
		16#440 : unicodeSymbol2cp866:=16#E0;
		16#441 : unicodeSymbol2cp866:=16#E1;
		16#442 : unicodeSymbol2cp866:=16#E2;
		16#443 : unicodeSymbol2cp866:=16#E3;
		16#444 : unicodeSymbol2cp866:=16#E4;
		16#445 : unicodeSymbol2cp866:=16#E5;
		16#446 : unicodeSymbol2cp866:=16#E6;
		16#447 : unicodeSymbol2cp866:=16#E7;
		16#448 : unicodeSymbol2cp866:=16#E8;
		16#449 : unicodeSymbol2cp866:=16#E9;
		16#44A : unicodeSymbol2cp866:=16#EA;
		16#44B : unicodeSymbol2cp866:=16#EB;
		16#44C : unicodeSymbol2cp866:=16#EC;
		16#44D : unicodeSymbol2cp866:=16#ED;
		16#44E : unicodeSymbol2cp866:=16#EE;
		16#44F : unicodeSymbol2cp866:=16#EF;
		16#401 : unicodeSymbol2cp866:=16#F0;
		16#451 : unicodeSymbol2cp866:=16#F1;
		16#404 : unicodeSymbol2cp866:=16#F2;
		16#454 : unicodeSymbol2cp866:=16#F3;
		16#407 : unicodeSymbol2cp866:=16#F4;
		16#457 : unicodeSymbol2cp866:=16#F5;
		16#40E : unicodeSymbol2cp866:=16#F6;
		16#45E : unicodeSymbol2cp866:=16#F7;
		16#B0 : unicodeSymbol2cp866:=16#F8;
		16#2219 : unicodeSymbol2cp866:=16#F9;
		16#B7 : unicodeSymbol2cp866:=16#FA;
		16#221A : unicodeSymbol2cp866:=16#FB;
		16#2116 : unicodeSymbol2cp866:=16#FC;
		16#A4 : unicodeSymbol2cp866:=16#FD;
		16#25A0 : unicodeSymbol2cp866:=16#FE;
		16#A0 : unicodeSymbol2cp866:=16#FF;
		ELSE
			unicodeSymbol2cp866:=16#3F; //?

END_CASE

END_FUNCTION

// CompWin/AppTerminalPost/DevCard/DeviceCard
PROGRAM DeviceCard
VAR
	crt: crt;
	lastCrtStatus: crtStatus;
	newCrtStatus: crtStatus;
	isInitialized: BOOL := FALSE;
	lockedTimer: TON;
	
	//CardID: STRING;
	CardType: EnumCardType := EnumCardType.UNDEFINED;
	_type: EnumCardType;
	
	// необходимость разблоикровки 
	_needLatchRelease: BOOL := TRUE;
END_VAR

//В самом начале с помощью метода init задаём конфигурацию модуля
//Это делается один раз
IF(NOT (isInitialized) AND PLC_PRG.comPortCard > 0)THEN
// инициализация картридера
	crt.init(iComPort := PLC_PRG.comPortCard);
	
	_needLatchRelease := TRUE;
	
	isInitialized :=  TRUE;
END_IF;

IF(isInitialized)THEN
	//проводим итерацию рабочего цикла и узнаём новый статус блока
	newCrtStatus := crt.iterateAndUpdateStatus();
	
	//Что либо проверять либо делать с блоком следует только когда он не занят
	IF newCrtStatus.error = CRT_NO_ERROR AND NOT(newCrtStatus.busy) THEN
		IF(newCrtStatus.cardState <> lastCrtStatus.cardState)THEN
			IF(newCrtStatus.cardState = CRT_RF_CARD_INSIDE) THEN
				//блок выполняется в момент вставления карты
				_type := GetTypeCard(cardId := crt.cardId);
				IF(_type <> EnumCardType.UNDEFINED)THEN
					crt.latchLock();
				ELSE
					//crt.latchRelease();
					_needLatchRelease := TRUE;
				END_IF; 
			ELSIF(newCrtStatus.cardState = CRT_NO_CARD)THEN
				 _type := EnumCardType.UNDEFINED;
				 //crt.latchRelease();
				 _needLatchRelease := TRUE;
			END_IF
		END_IF
		
		lastCrtStatus := newCrtStatus;
	
		// Если надо, то разблокировать карту
		IF(_needLatchRelease)THEN
			crt.latchRelease();
			_needLatchRelease := FALSE;
		END_IF 
	END_IF
	
	// реагировать на изменение типа карты
	IF(CardType <> _type)THEN
		CardType := _type;
		IF(NOT PLC_PRG.post.SetCard(_type, crt.cardId))THEN
			UnLockCard();
		END_IF
	END_IF	
END_IF

METHOD PUBLIC UnLockCard : BOOL
VAR_INPUT
END_VAR
// разблокировать карту
//crt.latchRelease();
_needLatchRelease := TRUE;

// отладка
DBG_PRG.UnLockCard();

//CardType := EnumCardType.UNDEFINED;
END_METHOD

METHOD PUBLIC DbgSetCard : BOOL
VAR_INPUT
END_VAR
//_type := DBG_PRG.debugStruct.CardType;
END_METHOD

METHOD PUBLIC GetTypeCard : EnumCardType
VAR_INPUT
	cardId : ARRAY [0..9] OF BYTE; // cardId первые 4 байта
END_VAR
VAR
	_arr: ARRAY[0..4] OF BYTE;
	_key: STRING;
	i: BYTE;
END_VAR
VAR CONSTANT
	// ключи уборки
	KEY_CLEANUP_COUNT: BYTE := 36;
	_kyesCleanup: ARRAY[0..KEY_CLEANUP_COUNT - 1] OF STRING := ['E58DCAE5', 'E5B3F3B0', '7D143C5B', 'DD133D5B', 'FDDC3B5B', '8DC73A5B', '74D72E0C', '0DCDB3A8', '32F9B3A8', '7B65B1A8', 
'9691B1A8', 'EE7AB1A8', '97B1B1A8', '99B8B1A8',
'D857B1A8',
'1834B1A8',
'077BB1A8',
// m9
'522BB4A8',
'D208B4A8',
'CA0FB4A8',
'13B12E02',//25-02-20
'23236102',//25-02-20 
//M10
 '0E1CB4A8',
 '22F8B3A8',
 'B9B6B3A8',
//M3 доп
'BDC43C5B',
//m11
 '1273B1A8',
 '1A8AB1A8',
 '5D98B1A8',
 //M2
 '0477B3DA',
//M12
'0427C3DA',
'4BDCB3A8',
'042DADDA',
//m6
 '04A5AEDA',
// M8 M9 05-12-2019
 '22D29622',
 '121C3534' // M8 26-07-2020
];
	
	// ключи инкассации
	KEY_CASHCOLLECT_COUNT: BYTE := 28;
	_kyesCashCollect: ARRAY[0..KEY_CASHCOLLECT_COUNT - 1] OF STRING := ['E42F290C', 'AD2C3A5B', '0D8C3C5B', '0DBB3B5B', '9DB63C5B', '559DCEE5', '15B3CCE5', '519BB3A8', '690CB4A8', '9CF9B3A8',
 'AF24B1A8', '2B9A7C38', '2CB6B1A8', '8D9DB1A8', 'CB5AB1A8', '4A2FB1A8',
'9230B1A8',
'031CB4A8',
'9492B1A8',
//m9
'032DB4A8',
'7AF6B3A8',
'23F9B3A8',
//M10
'5BBAB3A8',
'8EC8B3A8',
//M3 доп
'1D393C5B',

//M11
 '2B7FB1A8',
 '028FB1A8',
// M8 M9 05-12-2019
 '92AD5C35' 

];
	
	// ключи техслужбы
	KEY_SERVICE_COUNT: BYTE := 33;
	_kyesService: ARRAY[0..KEY_SERVICE_COUNT - 1] OF STRING := ['543A2F0C', '64EC250C', 'FDFC3A5B', '6D473D5B', 'AD603C5B', 'CD7A3A5B', '6533CAE5', 'D2F2B0A8', '070FB4A8', '7A1EB4A8', '200DB4A8',
 '5C48B1A8', 'C764B1A8', 'EE96B1A8', '4587B1A8', '0B9AB1A8',
'74B2B1A8',
'F6B4B1A8',
'9C28B1A8',
//m9
'E322B4A8',
'7515B4A8',
'C7C7B3A8',
//M10
'DAF7B3A8',
'FBA9B3A8',
//M3 доп
'EDB13B5B',

//M11
'19B8B1A8',
'38B1B1A8',

// M8, M9 VIP
'7578B1A8',
'D84EB1A8',
// M8 M9 05-12-2019
'633EE41A',
// M8 M9 11-03-2020
'7312BD03', // m88001 техника
'C3AF8B03',  // m89001 техника
// M8 26-07-2020
'E7F5B619' 



];
	
	// ключи добавления денег (бесплатной мойки)
	KEY_FREEMONEY_COUNT: BYTE := 3;
	_kyesFreeMoney: ARRAY[0..KEY_FREEMONEY_COUNT - 1] OF STRING := ['00000000', '559DCEE5', 'D643B1A8'];
END_VAR
GetTypeCard := EnumCardType.UNDEFINED;

// перевести занчение id  в строку ключа
_key := OSCAT_BASIC.BYTE_TO_STRH(cardId[0]);
_key := CONCAT(_key, OSCAT_BASIC.BYTE_TO_STRH(cardId[1]));
_key := CONCAT(_key, OSCAT_BASIC.BYTE_TO_STRH(cardId[2]));
_key := CONCAT(_key, OSCAT_BASIC.BYTE_TO_STRH(cardId[3]));

// Проверить ключи уборки
FOR i := 0 TO KEY_CLEANUP_COUNT - 1 DO
	IF(_key = _kyesCleanup[i])THEN
		EXIT;
	END_IF
END_FOR

IF(i < KEY_CLEANUP_COUNT)THEN
	GetTypeCard := EnumCardType.CLEANUP;
	RETURN;
END_IF

// Проверить ключи инкассации
FOR i := 0 TO KEY_CASHCOLLECT_COUNT - 1 DO
	IF(_key = _kyesCashCollect[i])THEN
		EXIT;
	END_IF
END_FOR

IF(i < KEY_CASHCOLLECT_COUNT)THEN
	GetTypeCard := EnumCardType.CASHCOLLECT;
	RETURN;
END_IF

// Проверить ключи техслужбы
FOR i := 0 TO KEY_SERVICE_COUNT - 1 DO
	IF(_key = _kyesService[i])THEN
		EXIT;
	END_IF
END_FOR

IF(i < KEY_SERVICE_COUNT)THEN
	GetTypeCard := EnumCardType.SERVICE;
	RETURN;
END_IF

// Проверить ключи добавления денег
FOR i := 0 TO KEY_FREEMONEY_COUNT - 1 DO
	IF(_key = _kyesFreeMoney[i])THEN
		EXIT;
	END_IF
END_FOR

IF(i < KEY_FREEMONEY_COUNT)THEN
	GetTypeCard := EnumCardType.FREEMONEY;
	RETURN;
END_IF
END_METHOD

METHOD TestValidComPort : BOOL
VAR_INPUT
	comPort: BYTE;
END_VAR
VAR
	maxnext: INT := 100;
	i: INT;
END_VAR
//TestValidComPort := FALSE;
//RETURN;

crt.init(iComPort := comPort);

newCrtStatus := crt.iterateAndUpdateStatus();

FOR i := 1 TO maxnext DO
	IF(not newCrtStatus.isInit) THEN
		newCrtStatus := crt.iterateAndUpdateStatus();
	ELSE
		EXIT;
	END_IF
END_FOR

//WHILE (newCrtStatus.busy) DO
//	newCrtStatus := crt.iterateAndUpdateStatus();
//END_WHILE

//newCrtStatus := crt.iterateAndUpdateStatus();

IF(newCrtStatus.error <> CRT_OPEN_ERROR)THEN
	TestValidComPort := TRUE;
ELSE
	TestValidComPort := FALSE;
END_IF

//IF newCrtStatus.error = CRT_NO_ERROR AND NOT(newCrtStatus.busy) THEN
//	TestValidComPort := TRUE;
//ELSE
//	TestValidComPort := FALSE;
//END_IF
END_METHOD

END_PROGRAM

// CompWin/AppTerminalPost/DevCard/crt
FUNCTION_BLOCK crt
VAR CONSTANT
	RESET_TRYCOUNT_DELAY : TIME := T#1000MS; //delay between reset tries	
	POLL_DELAY : TIME := T#200MS;
//	COM_PORT : BYTE := 2;  //use com2
	//commands consts
	CRT_INIT_COMMAND : crtParametrizedCommand := ( CM:= 16#30, PM := 16#31);	//init_and_lock_latch command
	CRT_STATUS_REQUEST_COMMAND : crtParametrizedCommand := ( CM:= 16#31, PM := 16#30); //status request command
	CRT_SERIAL_NUMBER_COMMAND : crtParametrizedCommand := ( CM:= 16#A2, PM:= 16#30);   //serial number command
    CRT_RF_CARD_RESET_COMMAND : crtParametrizedCommand := (CM:= 16#60, PM:=16#30);	   //rf card reset command
	CRT_LATCH_LOCK_COMMAND : crtParametrizedCommand := (CM:= 16#B0, PM:=16#30);	   //latch lock command
	CRT_LATCH_RELEASE_COMMAND : crtParametrizedCommand := (CM:= 16#B0, PM:=16#31);	   //latch release command
	CRT_RF_CARD_RESET_COMMAND_DATA : ARRAY [0..1] OF BYTE := [16#41, 16#42]; //set sequence OF rf card reset 
																			 //operation FOR different TYPE OF protocol Valid value: 41H (‘A’= Type A )，42H(‘B’= Type B ), 30H( ‘0’= Do not use)
			
	
	//program states:
	CRT_INIT_STATE : BYTE :=0;
	CRT_FATAL_ERROR  : BYTE :=1;
	CRT_DONE : BYTE := 3;
	CRT_RESET_STATE : BYTE := 4;
	CRT_DO_NOTHING : BYTE :=6;
	CRT_STATUS_REQUEST_STATE : BYTE := 7;
	CRT_RF_CARD_RESET : BYTE :=8;
	CRT_LOCK : BYTE :=9;
	CRT_RELEASE : BYTE :=10;
																			 
	CRT_CLOSE_COM_STATE : BYTE :=11;
END_VAR


VAR	

	//cachecode program states
	state : BYTE := CRT_INIT_STATE;
	
	error: CRT_ERROR := CRT_INIT_PROC_NOT_CALLED;
	
	lastCardState : CRT_CARD_STATE := CRT_CARD_UNDEFINED;
	newCardState : CRT_CARD_STATE ;
	
	locked : BOOL := FALSE;
	
	
	
	//com parameters
	crtComParams : ARRAY [1..7] OF COM.PARAMETER := [     
		(udiParameterId := COM.CAA_Parameter_Constants.udiPort, udiValue := 0),  // COM порт
		(udiParameterId := COM.CAA_Parameter_Constants.udiBaudrate, udiValue := 9600),
		(udiParameterId := COM.CAA_Parameter_Constants.udiParity,udiValue := INT_TO_UDINT(COM.PARITY.NONE)),
	    (udiParameterId := COM.CAA_Parameter_Constants.udiStopBits,udiValue := INT_TO_UDINT(COM.STOPBIT.ONESTOPBIT)),
		(udiParameterId := COM.CAA_Parameter_Constants.udiTimeout, udiValue := 0),
		(udiParameterId := COM.CAA_Parameter_Constants.udiByteSize, udiValue := 8),
		(udiParameterId := COM.CAA_Parameter_Constants.udiBinary,udiValue := 0)
	];
	
	crtOpen : COM.Open;
	crtClose : COM.Close;
	openedHCom : CAA.HANDLE := 0;
	portOpened : BOOL := FALSE;
	
	simpleCommand : crtSimpleCommand;
	
	
	
	waitTimer : TON;
	
	cardId : ARRAY [0..9] OF BYTE; // cardId первые 4 байта
	cardIdLen : BYTE :=0;
	b_crt_close_enable: BOOL := false;
END_VAR

METHOD init
VAR_INPUT
	iComPort: BYTE;
END_VAR
//init method called -> reset error flags
state := CRT_INIT_STATE;
//error := CRT_NO_ERROR;
error := CRT_OPEN_ERROR;

crtComParams[1].udiValue := iComPort;
END_METHOD

METHOD iterateAndUpdateStatus : crtStatus
//waiting between cycle
IF waitTimer.IN  THEN
	waitTimer(IN:= TRUE);
	IF NOT (waitTimer.Q) THEN
		iterateAndUpdateStatus.cardState := lastCardState;
		iterateAndUpdateStatus.busy := simpleCommand.xExecute;
		iterateAndUpdateStatus.locked := locked;
		iterateAndUpdateStatus.error := error;
		RETURN;
	ELSE
		waitTimer(IN:=FALSE);	
	END_IF
END_IF


CASE state OF
	CRT_INIT_STATE:
		crtOpen (xExecute := TRUE, 
				usiListLength := UINT_TO_USINT(SIZEOF(crtComParams)/SIZEOF(COM.PARAMETER)),
				pParameterList:= ADR(crtComParams)			
		);
		openedHCom := crtOpen.hCom;
		
		IF crtOpen.xError THEN
			crtOpen (xExecute := FALSE);
			portOpened := FALSE; 
			state := CRT_FATAL_ERROR;
			iterateAndUpdateStatus.isInit := TRUE;
			error := CRT_OPEN_ERROR;
		END_IF;
		
		IF crtOpen.xDone THEN
			crtOpen (xExecute := FALSE);
			portOpened := TRUE; 
			state := CRT_RESET_STATE;
			error := CRT_NO_ERROR;
 
		END_IF;
		
		IF(NOT crtOpen.xError AND crtOpen.xDone)THEN
			//simpleCommand(xExecute:=TRUE, hCom := crtOpen.hCom, xCommandDataSize:=0, xCommand:= CRT_INIT_COMMAND , xCommandDataSize:=0);
		
			//IF simpleCommand.xDone THEN
			//	error := CRT_NO_ERROR;
			//END_IF
		END_IF
		
	CRT_RESET_STATE:
		//initialize and release lock
		simpleCommand(xExecute:=TRUE, hCom := openedHCom, xCommandDataSize:=0, xCommand:= CRT_INIT_COMMAND , xCommandDataSize:=0);
		
		IF simpleCommand.xDone THEN

			iterateAndUpdateStatus.isInit := TRUE;
			IF(NOT simpleCommand.xError)THEN
				error := CRT_NO_ERROR;
			ELSE
				error := CRT_OPEN_ERROR;							
			END_IF

			newCardState := crtDecodeCardState(iST0:=simpleCommand.xST0, iST1:=simpleCommand.xST1);
			locked := (simpleCommand.xST1 = 16#30); 
			state := CRT_STATUS_REQUEST_STATE;
			waitTimer(IN:= TRUE, PT := RESET_TRYCOUNT_DELAY);
		END_IF
		
		//retry reset
		IF simpleCommand.xError THEN
			newCardState := CRT_CARD_UNDEFINED;    
			state := CRT_CLOSE_COM_STATE;
			//state := CRT_RESET_STATE;
			waitTimer(IN:= TRUE, PT := POLL_DELAY);
			
			//iterateAndUpdateStatus.isInit := TRUE;
			//error := CRT_OPEN_ERROR;			
		END_IF
		
